    movel([0.255095, -1.387885, -2.566810, -0.757694, 1.570796, 1.825892],accel_mss,speed_ms,0,blend_radius_m)
    movel([0.255265, -1.387620, -2.567000, -0.757769, 1.570796, 1.826062],accel_mss,speed_ms,0,blend_radius_m)
    movel([0.255538, -1.387474, -2.567104, -0.757811, 1.570796, 1.826334],accel_mss,speed_ms,0,blend_radius_m)
    movel([0.255936, -1.387475, -2.567104, -0.757810, 1.570796, 1.826733],accel_mss,speed_ms,0,blend_radius_m)
    movel([0.256466, -1.387632, -2.566991, -0.757766, 1.570796, 1.827262],accel_mss,speed_ms,0,blend_radius_m)
    movel([0.257289, -1.388179, -2.566600, -0.757611, 1.570796, 1.828085],accel_mss,speed_ms,0,blend_radius_m)
    movel([0.257855, -1.389086, -2.565949, -0.757354, 1.570796, 1.828651],accel_mss,speed_ms,0,blend_radius_m)
    movel([0.258263, -1.390555, -2.564893, -0.756941, 1.570796, 1.829060],accel_mss,speed_ms,0,blend_radius_m)
    movel([0.259108, -1.396147, -2.560843, -0.755399, 1.570796, 1.829904],accel_mss,speed_ms,0,blend_radius_m)
    movel([0.259420, -1.397275, -2.560021, -0.755093, 1.570796, 1.830216],accel_mss,speed_ms,0,blend_radius_m)
    movel([0.259859, -1.398329, -2.559250, -0.754809, 1.570796, 1.830656],accel_mss,speed_ms,0,blend_radius_m)
    movel([0.260330, -1.399097, -2.558688, -0.754603, 1.570796, 1.831126],accel_mss,speed_ms,0,blend_radius_m)
    movel([0.260925, -1.399770, -2.558195, -0.754424, 1.570796, 1.831721],accel_mss,speed_ms,0,blend_radius_m)
    movel([0.261593, -1.400274, -2.557826, -0.754290, 1.570796, 1.832390],accel_mss,speed_ms,0,blend_radius_m)
    movel([0.262390, -1.400639, -2.557557, -0.754193, 1.570796, 1.833187],accel_mss,speed_ms,0,blend_radius_m)
    movel([0.263557, -1.400866, -2.557390, -0.754133, 1.570796, 1.834353],accel_mss,speed_ms,0,blend_radius_m)
    movel([0.264871, -1.400801, -2.557438, -0.754150, 1.570796, 1.835667],accel_mss,speed_ms,0,blend_radius_m)
    movel([0.266400, -1.400447, -2.557698, -0.754244, 1.570796, 1.837196],accel_mss,speed_ms,0,blend_radius_m)
    movel([0.267947, -1.399865, -2.558125, -0.754398, 1.570796, 1.838744],accel_mss,speed_ms,0,blend_radius_m)
    movel([0.269799, -1.398926, -2.558813, -0.754649, 1.570796, 1.840596],accel_mss,speed_ms,0,blend_radius_m)
    movel([0.271593, -1.397805, -2.559633, -0.754950, 1.570796, 1.842389],accel_mss,speed_ms,0,blend_radius_m)
    movel([0.273718, -1.396265, -2.560757, -0.755367, 1.570796, 1.844514],accel_mss,speed_ms,0,blend_radius_m)
    movel([0.276733, -1.393794, -2.562553, -0.756042, 1.570796, 1.847530],accel_mss,speed_ms,0,blend_radius_m)
    movel([0.277800, -1.392821, -2.563257, -0.756311, 1.570796, 1.848596],accel_mss,speed_ms,0,blend_radius_m)
    movel([0.279582, -1.391076, -2.564517, -0.756796, 1.570796, 1.850378],accel_mss,speed_ms,0,blend_radius_m)
    movel([0.281480, -1.388952, -2.566045, -0.757392, 1.570796, 1.852277],accel_mss,speed_ms,0,blend_radius_m)
    movel([0.283244, -1.386754, -2.567620, -0.758016, 1.570796, 1.854040],accel_mss,speed_ms,0,blend_radius_m)
    movel([0.285091, -1.384211, -2.569432, -0.758746, 1.570796, 1.855887],accel_mss,speed_ms,0,blend_radius_m)
    movel([0.286815, -1.381625, -2.571266, -0.759499, 1.570796, 1.857611],accel_mss,speed_ms,0,blend_radius_m)
    movel([0.288428, -1.378981, -2.573130, -0.760278, 1.570796, 1.859225],accel_mss,speed_ms,0,blend_radius_m)
    movel([0.289908, -1.376305, -2.575007, -0.761077, 1.570796, 1.860704],accel_mss,speed_ms,0,blend_radius_m)
    movel([0.291098, -1.373867, -2.576709, -0.761814, 1.570796, 1.861894],accel_mss,speed_ms,0,blend_radius_m)
    movel([0.292109, -1.371416, -2.578410, -0.762563, 1.570796, 1.862906],accel_mss,speed_ms,0,blend_radius_m)
    movel([0.292732, -1.369549, -2.579701, -0.763139, 1.570796, 1.863528],accel_mss,speed_ms,0,blend_radius_m)
    movel([0.293193, -1.367698, -2.580975, -0.763716, 1.570796, 1.863989],accel_mss,speed_ms,0,blend_radius_m)
    movel([0.293453, -1.365997, -2.582142, -0.764250, 1.570796, 1.864249],accel_mss,speed_ms,0,blend_radius_m)
    movel([0.293523, -1.364348, -2.583270, -0.764771, 1.570796, 1.864319],accel_mss,speed_ms,0,blend_radius_m)
    movel([0.293397, -1.362735, -2.584369, -0.765285, 1.570796, 1.864193],accel_mss,speed_ms,0,blend_radius_m)
    movel([0.293080, -1.361208, -2.585406, -0.765775, 1.570796, 1.863876],accel_mss,speed_ms,0,blend_radius_m)
    movel([0.292542, -1.359616, -2.586484, -0.766289, 1.570796, 1.863339],accel_mss,speed_ms,0,blend_radius_m)
    movel([0.291851, -1.358116, -2.587496, -0.766777, 1.570796, 1.862647],accel_mss,speed_ms,0,blend_radius_m)
    movel([0.290674, -1.356227, -2.588766, -0.767395, 1.570796, 1.861471],accel_mss,speed_ms,0,blend_radius_m)
    movel([0.290146, -1.355630, -2.589167, -0.767592, 1.570796, 1.860942],accel_mss,speed_ms,0,blend_radius_m)
    movel([0.289507, -1.355132, -2.589501, -0.767756, 1.570796, 1.860303],accel_mss,speed_ms,0,blend_radius_m)
    movel([0.288952, -1.354872, -2.589675, -0.767843, 1.570796, 1.859748],accel_mss,speed_ms,0,blend_radius_m)
    movel([0.288300, -1.354741, -2.589762, -0.767886, 1.570796, 1.859097],accel_mss,speed_ms,0,blend_radius_m)
    movel([0.287679, -1.354781, -2.589735, -0.767872, 1.570796, 1.858476],accel_mss,speed_ms,0,blend_radius_m)
    movel([0.287015, -1.355005, -2.589585, -0.767798, 1.570796, 1.857811],accel_mss,speed_ms,0,blend_radius_m)
    movel([0.286082, -1.355625, -2.589170, -0.767594, 1.570796, 1.856878],accel_mss,speed_ms,0,blend_radius_m)
    movel([0.285289, -1.356517, -2.588572, -0.767300, 1.570796, 1.856086],accel_mss,speed_ms,0,blend_radius_m)
    movel([0.284369, -1.358039, -2.587548, -0.766802, 1.570796, 1.855165],accel_mss,speed_ms,0,blend_radius_m)
    movel([0.282752, -1.361200, -2.585411, -0.765777, 1.570796, 1.853548],accel_mss,speed_ms,0,blend_radius_m)
    movel([0.280629, -1.365085, -2.582766, -0.764537, 1.570796, 1.851426],accel_mss,speed_ms,0,blend_radius_m)
    movel([0.278252, -1.368753, -2.580249, -0.763386, 1.570796, 1.849048],accel_mss,speed_ms,0,blend_radius_m)
    movel([0.275849, -1.371892, -2.578080, -0.762416, 1.570796, 1.846645],accel_mss,speed_ms,0,blend_radius_m)
    movel([0.274806, -1.373052, -2.577275, -0.762062, 1.570796, 1.845602],accel_mss,speed_ms,0,blend_radius_m)
    movel([0.272903, -1.374773, -2.576077, -0.761539, 1.570796, 1.843700],accel_mss,speed_ms,0,blend_radius_m)
    movel([0.272221, -1.375292, -2.575715, -0.761382, 1.570796, 1.843017],accel_mss,speed_ms,0,blend_radius_m)
    movel([0.270902, -1.376104, -2.575148, -0.761137, 1.570796, 1.841698],accel_mss,speed_ms,0,blend_radius_m)
    movel([0.270153, -1.376475, -2.574888, -0.761026, 1.570796, 1.840949],accel_mss,speed_ms,0,blend_radius_m)
    movel([0.269154, -1.376784, -2.574672, -0.760933, 1.570796, 1.839950],accel_mss,speed_ms,0,blend_radius_m)
    movel([0.268438, -1.376865, -2.574615, -0.760909, 1.570796, 1.839235],accel_mss,speed_ms,0,blend_radius_m)
    movel([0.267352, -1.376877, -2.574607, -0.760905, 1.570796, 1.838149],accel_mss,speed_ms,0,blend_radius_m)
    movel([0.267003, -1.376777, -2.574677, -0.760935, 1.570796, 1.837799],accel_mss,speed_ms,0,blend_radius_m)
    movel([0.266387, -1.376391, -2.574947, -0.761051, 1.570796, 1.837183],accel_mss,speed_ms,0,blend_radius_m)
    movel([0.266133, -1.376115, -2.575140, -0.761134, 1.570796, 1.836929],accel_mss,speed_ms,0,blend_radius_m)
    movel([0.265758, -1.375526, -2.575552, -0.761311, 1.570796, 1.836554],accel_mss,speed_ms,0,blend_radius_m)
    movel([0.265630, -1.375043, -2.575889, -0.761457, 1.570796, 1.836426],accel_mss,speed_ms,0,blend_radius_m)
    movel([0.265067, -1.369773, -2.579546, -0.763070, 1.570796, 1.835863],accel_mss,speed_ms,0,blend_radius_m)
    movel([0.264692, -1.365521, -2.582468, -0.764400, 1.570796, 1.835488],accel_mss,speed_ms,0,blend_radius_m)
    movel([0.263976, -1.360329, -2.586002, -0.766058, 1.570796, 1.834772],accel_mss,speed_ms,0,blend_radius_m)
    movel([0.263461, -1.358019, -2.587561, -0.766808, 1.570796, 1.834258],accel_mss,speed_ms,0,blend_radius_m)
    movel([0.262803, -1.355819, -2.589040, -0.767530, 1.570796, 1.833599],accel_mss,speed_ms,0,blend_radius_m)
    movel([0.261961, -1.353719, -2.590445, -0.768225, 1.570796, 1.832758],accel_mss,speed_ms,0,blend_radius_m)
    movel([0.261016, -1.351955, -2.591621, -0.768813, 1.570796, 1.831812],accel_mss,speed_ms,0,blend_radius_m)
    movel([0.259856, -1.350343, -2.592692, -0.769355, 1.570796, 1.830652],accel_mss,speed_ms,0,blend_radius_m)
    movel([0.258562, -1.348990, -2.593587, -0.769812, 1.570796, 1.829358],accel_mss,speed_ms,0,blend_radius_m)
    movel([0.257068, -1.347816, -2.594362, -0.770211, 1.570796, 1.827864],accel_mss,speed_ms,0,blend_radius_m)
    movel([0.255389, -1.346838, -2.595007, -0.770544, 1.570796, 1.826185],accel_mss,speed_ms,0,blend_radius_m)
    movel([0.253535, -1.346063, -2.595516, -0.770810, 1.570796, 1.824331],accel_mss,speed_ms,0,blend_radius_m)
    movel([0.252415, -1.345708, -2.595749, -0.770932, 1.570796, 1.823211],accel_mss,speed_ms,0,blend_radius_m)
    movel([0.251733, -1.345613, -2.595812, -0.770964, 1.570796, 1.822529],accel_mss,speed_ms,0,blend_radius_m)
    movel([0.251230, -1.345713, -2.595746, -0.770930, 1.570796, 1.822027],accel_mss,speed_ms,0,blend_radius_m)
    movel([0.250768, -1.346010, -2.595551, -0.770828, 1.570796, 1.821565],accel_mss,speed_ms,0,blend_radius_m)
    movel([0.250318, -1.346670, -2.595117, -0.770602, 1.570796, 1.821115],accel_mss,speed_ms,0,blend_radius_m)
    movel([0.249924, -1.348002, -2.594240, -0.770147, 1.570796, 1.820721],accel_mss,speed_ms,0,blend_radius_m)
    movel([0.249536, -1.349939, -2.592959, -0.769491, 1.570796, 1.820333],accel_mss,speed_ms,0,blend_radius_m)
    movel([0.249117, -1.352828, -2.591040, -0.768521, 1.570796, 1.819913],accel_mss,speed_ms,0,blend_radius_m)
    movel([0.248523, -1.356486, -2.588593, -0.767310, 1.570796, 1.819319],accel_mss,speed_ms,0,blend_radius_m)
    movel([0.248092, -1.358275, -2.587389, -0.766725, 1.570796, 1.818888],accel_mss,speed_ms,0,blend_radius_m)
    movel([0.246220, -1.365023, -2.582809, -0.764557, 1.570796, 1.817017],accel_mss,speed_ms,0,blend_radius_m)
    movel([0.245321, -1.367822, -2.580890, -0.763677, 1.570796, 1.816117],accel_mss,speed_ms,0,blend_radius_m)
    movel([0.242201, -1.375991, -2.575227, -0.761171, 1.570796, 1.812997],accel_mss,speed_ms,0,blend_radius_m)
    movel([0.239764, -1.381897, -2.571073, -0.759419, 1.570796, 1.810560],accel_mss,speed_ms,0,blend_radius_m)
    movel([0.237387, -1.387154, -2.567333, -0.757902, 1.570796, 1.808183],accel_mss,speed_ms,0,blend_radius_m)
    movel([0.235039, -1.391842, -2.563965, -0.756582, 1.570796, 1.805836],accel_mss,speed_ms,0,blend_radius_m)
    movel([0.231786, -1.397514, -2.559846, -0.755029, 1.570796, 1.802583],accel_mss,speed_ms,0,blend_radius_m)
    movel([0.231472, -1.397972, -2.559512, -0.754905, 1.570796, 1.802268],accel_mss,speed_ms,0,blend_radius_m)
    movel([0.231229, -1.398184, -2.559356, -0.754848, 1.570796, 1.802025],accel_mss,speed_ms,0,blend_radius_m)
    movel([0.230929, -1.398295, -2.559276, -0.754818, 1.570796, 1.801725],accel_mss,speed_ms,0,blend_radius_m)
    movel([0.230719, -1.398272, -2.559292, -0.754825, 1.570796, 1.801515],accel_mss,speed_ms,0,blend_radius_m)
    movel([0.230647, -1.398140, -2.559389, -0.754860, 1.570796, 1.801444],accel_mss,speed_ms,0,blend_radius_m)
    movel([0.231423, -1.395310, -2.561452, -0.755627, 1.570796, 1.802219],accel_mss,speed_ms,0,blend_radius_m)
    movel([0.231535, -1.394305, -2.562182, -0.755902, 1.570796, 1.802332],accel_mss,speed_ms,0,blend_radius_m)
    movel([0.231433, -1.393186, -2.562993, -0.756210, 1.570796, 1.802229],accel_mss,speed_ms,0,blend_radius_m)
    movel([0.231036, -1.391255, -2.564388, -0.756746, 1.570796, 1.801833],accel_mss,speed_ms,0,blend_radius_m)
    movel([0.230646, -1.388956, -2.566042, -0.757391, 1.570796, 1.801443],accel_mss,speed_ms,0,blend_radius_m)
    movel([0.230572, -1.386887, -2.567524, -0.757978, 1.570796, 1.801369],accel_mss,speed_ms,0,blend_radius_m)
    movel([0.230812, -1.384183, -2.569452, -0.758754, 1.570796, 1.801608],accel_mss,speed_ms,0,blend_radius_m)
    movel([0.231528, -1.379286, -2.572916, -0.760188, 1.570796, 1.802324],accel_mss,speed_ms,0,blend_radius_m)
    movel([0.232292, -1.373125, -2.577225, -0.762040, 1.570796, 1.803089],accel_mss,speed_ms,0,blend_radius_m)
    movel([0.232470, -1.370485, -2.579054, -0.762850, 1.570796, 1.803266],accel_mss,speed_ms,0,blend_radius_m)
    movel([0.232513, -1.367882, -2.580849, -0.763658, 1.570796, 1.803309],accel_mss,speed_ms,0,blend_radius_m)
    movel([0.232417, -1.365596, -2.582417, -0.764376, 1.570796, 1.803213],accel_mss,speed_ms,0,blend_radius_m)
    movel([0.232184, -1.363359, -2.583944, -0.765086, 1.570796, 1.802980],accel_mss,speed_ms,0,blend_radius_m)
    movel([0.231819, -1.361328, -2.585325, -0.765736, 1.570796, 1.802616],accel_mss,speed_ms,0,blend_radius_m)
    movel([0.231292, -1.359376, -2.586646, -0.766367, 1.570796, 1.802088],accel_mss,speed_ms,0,blend_radius_m)
    movel([0.230545, -1.357337, -2.588021, -0.767031, 1.570796, 1.801342],accel_mss,speed_ms,0,blend_radius_m)
    movel([0.229699, -1.355644, -2.589158, -0.767588, 1.570796, 1.800495],accel_mss,speed_ms,0,blend_radius_m)
    movel([0.228650, -1.354120, -2.590177, -0.768091, 1.570796, 1.799447],accel_mss,speed_ms,0,blend_radius_m)
    movel([0.227292, -1.352590, -2.591198, -0.768601, 1.570796, 1.798088],accel_mss,speed_ms,0,blend_radius_m)
    movel([0.225840, -1.351336, -2.592032, -0.769021, 1.570796, 1.796636],accel_mss,speed_ms,0,blend_radius_m)
    movel([0.224294, -1.350424, -2.592638, -0.769327, 1.570796, 1.795090],accel_mss,speed_ms,0,blend_radius_m)
    movel([0.222638, -1.349849, -2.593019, -0.769521, 1.570796, 1.793435],accel_mss,speed_ms,0,blend_radius_m)
    movel([0.220857, -1.349600, -2.593184, -0.769605, 1.570796, 1.791653],accel_mss,speed_ms,0,blend_radius_m)
    movel([0.219370, -1.349643, -2.593155, -0.769591, 1.570796, 1.790166],accel_mss,speed_ms,0,blend_radius_m)
    movel([0.217805, -1.349909, -2.592979, -0.769501, 1.570796, 1.788601],accel_mss,speed_ms,0,blend_radius_m)
    movel([0.216251, -1.350382, -2.592666, -0.769342, 1.570796, 1.787048],accel_mss,speed_ms,0,blend_radius_m)
    movel([0.214697, -1.351068, -2.592211, -0.769111, 1.570796, 1.785493],accel_mss,speed_ms,0,blend_radius_m)
    movel([0.213185, -1.351948, -2.591625, -0.768815, 1.570796, 1.783981],accel_mss,speed_ms,0,blend_radius_m)
    movel([0.211756, -1.352999, -2.590926, -0.768464, 1.570796, 1.782553],accel_mss,speed_ms,0,blend_radius_m)
    movel([0.210399, -1.354224, -2.590108, -0.768057, 1.570796, 1.781195],accel_mss,speed_ms,0,blend_radius_m)
    movel([0.208813, -1.356025, -2.588902, -0.767462, 1.570796, 1.779609],accel_mss,speed_ms,0,blend_radius_m)
    movel([0.208461, -1.356503, -2.588581, -0.767305, 1.570796, 1.779257],accel_mss,speed_ms,0,blend_radius_m)
    movel([0.207795, -1.357594, -2.587848, -0.766947, 1.570796, 1.778591],accel_mss,speed_ms,0,blend_radius_m)
    movel([0.207515, -1.357910, -2.587635, -0.766844, 1.570796, 1.778311],accel_mss,speed_ms,0,blend_radius_m)
    movel([0.207218, -1.358097, -2.587509, -0.766783, 1.570796, 1.778014],accel_mss,speed_ms,0,blend_radius_m)
    movel([0.206945, -1.358140, -2.587480, -0.766769, 1.570796, 1.777741],accel_mss,speed_ms,0,blend_radius_m)
    movel([0.206737, -1.357986, -2.587584, -0.766819, 1.570796, 1.777533],accel_mss,speed_ms,0,blend_radius_m)
    movel([0.206764, -1.357690, -2.587783, -0.766916, 1.570796, 1.777560],accel_mss,speed_ms,0,blend_radius_m)
    movel([0.207503, -1.356392, -2.588655, -0.767341, 1.570796, 1.778299],accel_mss,speed_ms,0,blend_radius_m)
    movel([0.208775, -1.354760, -2.589750, -0.767879, 1.570796, 1.779572],accel_mss,speed_ms,0,blend_radius_m)
    movel([0.210327, -1.353184, -2.590803, -0.768403, 1.570796, 1.781123],accel_mss,speed_ms,0,blend_radius_m)
    movel([0.211548, -1.352151, -2.591491, -0.768748, 1.570796, 1.782344],accel_mss,speed_ms,0,blend_radius_m)
    movel([0.212843, -1.351218, -2.592111, -0.769060, 1.570796, 1.783639],accel_mss,speed_ms,0,blend_radius_m)
    movel([0.214163, -1.350420, -2.592640, -0.769329, 1.570796, 1.784959],accel_mss,speed_ms,0,blend_radius_m)
    movel([0.215522, -1.349753, -2.593082, -0.769554, 1.570796, 1.786318],accel_mss,speed_ms,0,blend_radius_m)
    movel([0.216900, -1.349227, -2.593431, -0.769732, 1.570796, 1.787696],accel_mss,speed_ms,0,blend_radius_m)
    movel([0.218268, -1.348854, -2.593677, -0.769858, 1.570796, 1.789065],accel_mss,speed_ms,0,blend_radius_m)
    movel([0.219652, -1.348624, -2.593829, -0.769936, 1.570796, 1.790448],accel_mss,speed_ms,0,blend_radius_m)
    movel([0.220986, -1.348545, -2.593881, -0.769963, 1.570796, 1.791782],accel_mss,speed_ms,0,blend_radius_m)
    movel([0.222782, -1.348704, -2.593776, -0.769909, 1.570796, 1.793578],accel_mss,speed_ms,0,blend_radius_m)
    movel([0.224379, -1.349179, -2.593462, -0.769748, 1.570796, 1.795175],accel_mss,speed_ms,0,blend_radius_m)
    movel([0.226051, -1.350036, -2.592895, -0.769458, 1.570796, 1.796847],accel_mss,speed_ms,0,blend_radius_m)
    movel([0.227532, -1.351097, -2.592191, -0.769101, 1.570796, 1.798328],accel_mss,speed_ms,0,blend_radius_m)
    movel([0.228968, -1.352491, -2.591264, -0.768634, 1.570796, 1.799764],accel_mss,speed_ms,0,blend_radius_m)
    movel([0.230183, -1.354068, -2.590212, -0.768109, 1.570796, 1.800979],accel_mss,speed_ms,0,blend_radius_m)
    movel([0.231241, -1.355893, -2.588990, -0.767505, 1.570796, 1.802037],accel_mss,speed_ms,0,blend_radius_m)
    movel([0.232082, -1.357856, -2.587671, -0.766862, 1.570796, 1.802878],accel_mss,speed_ms,0,blend_radius_m)
    movel([0.232741, -1.360024, -2.586208, -0.766157, 1.570796, 1.803537],accel_mss,speed_ms,0,blend_radius_m)
    movel([0.233194, -1.362294, -2.584669, -0.765426, 1.570796, 1.803990],accel_mss,speed_ms,0,blend_radius_m)
    movel([0.233471, -1.364806, -2.582957, -0.764626, 1.570796, 1.804267],accel_mss,speed_ms,0,blend_radius_m)
    movel([0.233565, -1.367384, -2.581191, -0.763814, 1.570796, 1.804361],accel_mss,speed_ms,0,blend_radius_m)
    movel([0.233479, -1.370501, -2.579043, -0.762845, 1.570796, 1.804275],accel_mss,speed_ms,0,blend_radius_m)
    movel([0.233220, -1.373662, -2.576851, -0.761876, 1.570796, 1.804017],accel_mss,speed_ms,0,blend_radius_m)
    movel([0.232141, -1.381784, -2.571153, -0.759452, 1.570796, 1.802937],accel_mss,speed_ms,0,blend_radius_m)
    movel([0.231723, -1.384753, -2.569046, -0.758590, 1.570796, 1.802520],accel_mss,speed_ms,0,blend_radius_m)
    movel([0.231587, -1.386705, -2.567654, -0.758030, 1.570796, 1.802384],accel_mss,speed_ms,0,blend_radius_m)
    movel([0.231680, -1.388416, -2.566430, -0.757543, 1.570796, 1.802476],accel_mss,speed_ms,0,blend_radius_m)
    movel([0.232016, -1.390502, -2.564931, -0.756956, 1.570796, 1.802813],accel_mss,speed_ms,0,blend_radius_m)
    movel([0.232538, -1.393687, -2.562630, -0.756072, 1.570796, 1.803334],accel_mss,speed_ms,0,blend_radius_m)
    movel([0.232642, -1.394026, -2.562384, -0.755978, 1.570796, 1.803438],accel_mss,speed_ms,0,blend_radius_m)
    movel([0.232836, -1.393978, -2.562419, -0.755992, 1.570796, 1.803633],accel_mss,speed_ms,0,blend_radius_m)
    movel([0.233230, -1.393353, -2.562872, -0.756164, 1.570796, 1.804026],accel_mss,speed_ms,0,blend_radius_m)
    movel([0.237057, -1.385694, -2.568376, -0.758319, 1.570796, 1.807853],accel_mss,speed_ms,0,blend_radius_m)
    movel([0.239796, -1.379520, -2.572750, -0.760118, 1.570796, 1.810592],accel_mss,speed_ms,0,blend_radius_m)
    movel([0.242407, -1.373049, -2.577278, -0.762063, 1.570796, 1.813204],accel_mss,speed_ms,0,blend_radius_m)
    movel([0.244761, -1.366579, -2.581744, -0.764067, 1.570796, 1.815557],accel_mss,speed_ms,0,blend_radius_m)
    movel([0.245773, -1.363351, -2.583950, -0.765088, 1.570796, 1.816569],accel_mss,speed_ms,0,blend_radius_m)
    movel([0.246728, -1.359698, -2.586428, -0.766263, 1.570796, 1.817525],accel_mss,speed_ms,0,blend_radius_m)
    movel([0.247527, -1.356058, -2.588880, -0.767451, 1.570796, 1.818323],accel_mss,speed_ms,0,blend_radius_m)
    movel([0.248051, -1.352879, -2.591005, -0.768504, 1.570796, 1.818848],accel_mss,speed_ms,0,blend_radius_m)
    movel([0.248446, -1.350238, -2.592761, -0.769390, 1.570796, 1.819242],accel_mss,speed_ms,0,blend_radius_m)
    movel([0.248857, -1.348235, -2.594086, -0.770068, 1.570796, 1.819653],accel_mss,speed_ms,0,blend_radius_m)
    movel([0.249288, -1.346744, -2.595068, -0.770577, 1.570796, 1.820084],accel_mss,speed_ms,0,blend_radius_m)
    movel([0.249754, -1.345882, -2.595635, -0.770872, 1.570796, 1.820550],accel_mss,speed_ms,0,blend_radius_m)
    movel([0.250249, -1.345323, -2.596002, -0.771064, 1.570796, 1.821045],accel_mss,speed_ms,0,blend_radius_m)
    movel([0.250776, -1.344913, -2.596271, -0.771205, 1.570796, 1.821572],accel_mss,speed_ms,0,blend_radius_m)
    movel([0.251321, -1.344661, -2.596436, -0.771292, 1.570796, 1.822117],accel_mss,speed_ms,0,blend_radius_m)
    movel([0.251873, -1.344569, -2.596497, -0.771324, 1.570796, 1.822669],accel_mss,speed_ms,0,blend_radius_m)
    movel([0.252588, -1.344649, -2.596444, -0.771296, 1.570796, 1.823385],accel_mss,speed_ms,0,blend_radius_m)
    movel([0.253955, -1.345029, -2.596195, -0.771165, 1.570796, 1.824751],accel_mss,speed_ms,0,blend_radius_m)
    movel([0.256341, -1.345925, -2.595607, -0.770857, 1.570796, 1.827138],accel_mss,speed_ms,0,blend_radius_m)
    movel([0.258315, -1.347164, -2.594792, -0.770433, 1.570796, 1.829111],accel_mss,speed_ms,0,blend_radius_m)
    movel([0.260118, -1.348786, -2.593722, -0.769881, 1.570796, 1.830914],accel_mss,speed_ms,0,blend_radius_m)
    movel([0.261674, -1.350714, -2.592445, -0.769230, 1.570796, 1.832470],accel_mss,speed_ms,0,blend_radius_m)
    movel([0.262915, -1.352863, -2.591016, -0.768509, 1.570796, 1.833711],accel_mss,speed_ms,0,blend_radius_m)
    movel([0.263612, -1.354489, -2.589931, -0.767969, 1.570796, 1.834408],accel_mss,speed_ms,0,blend_radius_m)
    movel([0.264185, -1.356184, -2.588795, -0.767410, 1.570796, 1.834981],accel_mss,speed_ms,0,blend_radius_m)
    movel([0.265108, -1.360143, -2.586127, -0.766118, 1.570796, 1.835905],accel_mss,speed_ms,0,blend_radius_m)
    movel([0.265810, -1.365284, -2.582630, -0.764475, 1.570796, 1.836606],accel_mss,speed_ms,0,blend_radius_m)
    movel([0.266385, -1.372378, -2.577743, -0.762268, 1.570796, 1.837182],accel_mss,speed_ms,0,blend_radius_m)
    movel([0.266613, -1.374304, -2.576404, -0.761681, 1.570796, 1.837409],accel_mss,speed_ms,0,blend_radius_m)
    movel([0.266771, -1.374866, -2.576012, -0.761511, 1.570796, 1.837568],accel_mss,speed_ms,0,blend_radius_m)
    movel([0.267041, -1.375360, -2.575667, -0.761361, 1.570796, 1.837837],accel_mss,speed_ms,0,blend_radius_m)
    movel([0.267347, -1.375658, -2.575460, -0.761272, 1.570796, 1.838143],accel_mss,speed_ms,0,blend_radius_m)
    movel([0.267760, -1.375844, -2.575329, -0.761215, 1.570796, 1.838556],accel_mss,speed_ms,0,blend_radius_m)
    movel([0.268285, -1.375927, -2.575272, -0.761191, 1.570796, 1.839082],accel_mss,speed_ms,0,blend_radius_m)
    movel([0.268867, -1.375899, -2.575291, -0.761199, 1.570796, 1.839663],accel_mss,speed_ms,0,blend_radius_m)
    movel([0.269616, -1.375740, -2.575402, -0.761247, 1.570796, 1.840412],accel_mss,speed_ms,0,blend_radius_m)
    movel([0.270377, -1.375462, -2.575596, -0.761331, 1.570796, 1.841174],accel_mss,speed_ms,0,blend_radius_m)
    movel([0.271129, -1.375077, -2.575865, -0.761447, 1.570796, 1.841925],accel_mss,speed_ms,0,blend_radius_m)
    movel([0.271844, -1.374596, -2.576200, -0.761592, 1.570796, 1.842640],accel_mss,speed_ms,0,blend_radius_m)
    movel([0.273576, -1.373133, -2.577219, -0.762037, 1.570796, 1.844373],accel_mss,speed_ms,0,blend_radius_m)
    movel([0.275126, -1.371513, -2.578343, -0.762533, 1.570796, 1.845922],accel_mss,speed_ms,0,blend_radius_m)
    movel([0.276981, -1.369177, -2.579957, -0.763255, 1.570796, 1.847777],accel_mss,speed_ms,0,blend_radius_m)
    movel([0.278604, -1.366757, -2.581622, -0.764011, 1.570796, 1.849400],accel_mss,speed_ms,0,blend_radius_m)
    movel([0.280459, -1.363589, -2.583787, -0.765012, 1.570796, 1.851256],accel_mss,speed_ms,0,blend_radius_m)
    movel([0.283390, -1.357989, -2.587582, -0.766818, 1.570796, 1.854186],accel_mss,speed_ms,0,blend_radius_m)
    movel([0.284147, -1.356672, -2.588468, -0.767249, 1.570796, 1.854944],accel_mss,speed_ms,0,blend_radius_m)
    movel([0.284772, -1.355802, -2.589051, -0.767535, 1.570796, 1.855569],accel_mss,speed_ms,0,blend_radius_m)
    movel([0.285460, -1.355101, -2.589521, -0.767767, 1.570796, 1.856256],accel_mss,speed_ms,0,blend_radius_m)
    movel([0.286130, -1.354583, -2.589868, -0.767938, 1.570796, 1.856926],accel_mss,speed_ms,0,blend_radius_m)
    movel([0.286753, -1.354223, -2.590108, -0.768057, 1.570796, 1.857549],accel_mss,speed_ms,0,blend_radius_m)
    movel([0.287401, -1.353985, -2.590268, -0.768136, 1.570796, 1.858197],accel_mss,speed_ms,0,blend_radius_m)
    movel([0.288149, -1.353838, -2.590366, -0.768185, 1.570796, 1.858946],accel_mss,speed_ms,0,blend_radius_m)
    movel([0.288852, -1.353812, -2.590383, -0.768194, 1.570796, 1.859649],accel_mss,speed_ms,0,blend_radius_m)
    movel([0.289487, -1.353922, -2.590310, -0.768157, 1.570796, 1.860283],accel_mss,speed_ms,0,blend_radius_m)
    movel([0.290701, -1.354530, -2.589903, -0.767956, 1.570796, 1.861497],accel_mss,speed_ms,0,blend_radius_m)
    movel([0.291837, -1.355686, -2.589129, -0.767574, 1.570796, 1.862634],accel_mss,speed_ms,0,blend_radius_m)
    movel([0.292934, -1.357455, -2.587941, -0.766993, 1.570796, 1.863730],accel_mss,speed_ms,0,blend_radius_m)
    movel([0.293974, -1.359880, -2.586306, -0.766204, 1.570796, 1.864770],accel_mss,speed_ms,0,blend_radius_m)
    movel([0.294523, -1.362239, -2.584706, -0.765444, 1.570796, 1.865319],accel_mss,speed_ms,0,blend_radius_m)
    movel([0.294624, -1.363458, -2.583877, -0.765054, 1.570796, 1.865420],accel_mss,speed_ms,0,blend_radius_m)
    movel([0.294609, -1.364722, -2.583014, -0.764653, 1.570796, 1.865406],accel_mss,speed_ms,0,blend_radius_m)
    movel([0.294266, -1.367507, -2.581107, -0.763775, 1.570796, 1.865062],accel_mss,speed_ms,0,blend_radius_m)
    movel([0.293918, -1.368891, -2.580154, -0.763344, 1.570796, 1.864714],accel_mss,speed_ms,0,blend_radius_m)
    movel([0.293268, -1.370843, -2.578807, -0.762739, 1.570796, 1.864064],accel_mss,speed_ms,0,blend_radius_m)
    movel([0.291751, -1.374603, -2.576196, -0.761590, 1.570796, 1.862547],accel_mss,speed_ms,0,blend_radius_m)
    movel([0.290553, -1.376888, -2.574599, -0.760902, 1.570796, 1.861349],accel_mss,speed_ms,0,blend_radius_m)
    speed_ms = 0.005
    movel([0.290553, -1.368165, -2.570582, -0.773641, 1.570796, 1.861349],accel_mss,speed_ms,0,blend_radius_m)
    speed_ms = 0.040
    movel([0.320654, -1.348290, -2.584044, -0.780055, 1.570796, 1.891451],accel_mss,speed_ms,0,blend_radius_m)
    speed_ms = 0.005
    movel([0.320654, -1.357148, -2.588148, -0.767093, 1.570796, 1.891451],accel_mss,speed_ms,0,blend_radius_m)
    speed_ms = 0.025
    movel([0.319732, -1.357074, -2.588198, -0.767118, 1.570796, 1.890528],accel_mss,speed_ms,0,blend_radius_m)
    movel([0.319205, -1.356915, -2.588304, -0.767170, 1.570796, 1.890001],accel_mss,speed_ms,0,blend_radius_m)
    movel([0.317857, -1.356295, -2.588721, -0.767373, 1.570796, 1.888654],accel_mss,speed_ms,0,blend_radius_m)
    movel([0.317320, -1.355922, -2.588971, -0.767496, 1.570796, 1.888117],accel_mss,speed_ms,0,blend_radius_m)
    movel([0.316201, -1.354707, -2.589785, -0.767897, 1.570796, 1.886997],accel_mss,speed_ms,0,blend_radius_m)
    movel([0.314823, -1.352667, -2.591147, -0.768575, 1.570796, 1.885619],accel_mss,speed_ms,0,blend_radius_m)
    movel([0.313237, -1.349704, -2.593115, -0.769570, 1.570796, 1.884034],accel_mss,speed_ms,0,blend_radius_m)
    movel([0.311845, -1.346731, -2.595077, -0.770581, 1.570796, 1.882641],accel_mss,speed_ms,0,blend_radius_m)
    movel([0.311446, -1.345137, -2.596124, -0.771128, 1.570796, 1.882243],accel_mss,speed_ms,0,blend_radius_m)
    movel([0.311462, -1.344439, -2.596581, -0.771368, 1.570796, 1.882258],accel_mss,speed_ms,0,blend_radius_m)
    movel([0.312033, -1.342330, -2.597959, -0.772099, 1.570796, 1.882830],accel_mss,speed_ms,0,blend_radius_m)
    movel([0.313181, -1.338985, -2.600133, -0.773272, 1.570796, 1.883977],accel_mss,speed_ms,0,blend_radius_m)
    movel([0.315208, -1.333366, -2.603748, -0.775275, 1.570796, 1.886004],accel_mss,speed_ms,0,blend_radius_m)
    movel([0.316058, -1.331299, -2.605067, -0.776022, 1.570796, 1.886855],accel_mss,speed_ms,0,blend_radius_m)
    movel([0.317881, -1.327107, -2.607725, -0.777556, 1.570796, 1.888677],accel_mss,speed_ms,0,blend_radius_m)
    movel([0.318194, -1.326115, -2.608351, -0.777923, 1.570796, 1.888990],accel_mss,speed_ms,0,blend_radius_m)
    movel([0.318267, -1.325423, -2.608786, -0.778179, 1.570796, 1.889064],accel_mss,speed_ms,0,blend_radius_m)
    movel([0.318110, -1.324962, -2.609077, -0.778351, 1.570796, 1.888907],accel_mss,speed_ms,0,blend_radius_m)
    movel([0.317737, -1.324753, -2.609207, -0.778428, 1.570796, 1.888533],accel_mss,speed_ms,0,blend_radius_m)
    movel([0.317436, -1.324772, -2.609196, -0.778421, 1.570796, 1.888233],accel_mss,speed_ms,0,blend_radius_m)
    movel([0.316115, -1.325001, -2.609052, -0.778336, 1.570796, 1.886911],accel_mss,speed_ms,0,blend_radius_m)
    movel([0.315993, -1.324904, -2.609113, -0.778372, 1.570796, 1.886790],accel_mss,speed_ms,0,blend_radius_m)
    movel([0.315921, -1.324400, -2.609429, -0.778560, 1.570796, 1.886717],accel_mss,speed_ms,0,blend_radius_m)
    movel([0.315980, -1.324129, -2.609599, -0.778661, 1.570796, 1.886777],accel_mss,speed_ms,0,blend_radius_m)
    movel([0.317198, -1.321892, -2.610999, -0.779498, 1.570796, 1.887995],accel_mss,speed_ms,0,blend_radius_m)
    movel([0.317469, -1.321421, -2.611293, -0.779675, 1.570796, 1.888265],accel_mss,speed_ms,0,blend_radius_m)
    movel([0.318083, -1.320351, -2.611960, -0.780079, 1.570796, 1.888879],accel_mss,speed_ms,0,blend_radius_m)
    movel([0.315622, -1.322333, -2.610723, -0.779332, 1.570796, 1.886419],accel_mss,speed_ms,0,blend_radius_m)
    movel([0.313339, -1.324104, -2.609615, -0.778670, 1.570796, 1.884135],accel_mss,speed_ms,0,blend_radius_m)
    movel([0.310995, -1.325778, -2.608563, -0.778048, 1.570796, 1.881791],accel_mss,speed_ms,0,blend_radius_m)
    movel([0.308638, -1.327328, -2.607586, -0.777475, 1.570796, 1.879434],accel_mss,speed_ms,0,blend_radius_m)
    movel([0.306302, -1.328723, -2.606703, -0.776962, 1.570796, 1.877099],accel_mss,speed_ms,0,blend_radius_m)
    movel([0.304835, -1.329490, -2.606218, -0.776682, 1.570796, 1.875632],accel_mss,speed_ms,0,blend_radius_m)
    movel([0.304548, -1.329552, -2.606178, -0.776659, 1.570796, 1.875345],accel_mss,speed_ms,0,blend_radius_m)
    movel([0.304344, -1.329458, -2.606238, -0.776693, 1.570796, 1.875141],accel_mss,speed_ms,0,blend_radius_m)
    movel([0.304305, -1.329242, -2.606375, -0.776772, 1.570796, 1.875101],accel_mss,speed_ms,0,blend_radius_m)
    movel([0.304442, -1.328987, -2.606536, -0.776866, 1.570796, 1.875238],accel_mss,speed_ms,0,blend_radius_m)
    movel([0.305573, -1.327819, -2.607276, -0.777294, 1.570796, 1.876370],accel_mss,speed_ms,0,blend_radius_m)
    movel([0.307878, -1.325397, -2.608803, -0.778189, 1.570796, 1.878674],accel_mss,speed_ms,0,blend_radius_m)
    movel([0.308860, -1.324183, -2.609565, -0.778641, 1.570796, 1.879657],accel_mss,speed_ms,0,blend_radius_m)
    movel([0.310446, -1.321890, -2.611000, -0.779499, 1.570796, 1.881243],accel_mss,speed_ms,0,blend_radius_m)
    movel([0.310222, -1.321875, -2.611010, -0.779504, 1.570796, 1.881019],accel_mss,speed_ms,0,blend_radius_m)
    movel([0.308575, -1.323006, -2.610303, -0.779080, 1.570796, 1.879372],accel_mss,speed_ms,0,blend_radius_m)
    movel([0.301104, -1.327684, -2.607361, -0.777344, 1.570796, 1.871900],accel_mss,speed_ms,0,blend_radius_m)
    movel([0.299050, -1.329068, -2.606485, -0.776836, 1.570796, 1.869847],accel_mss,speed_ms,0,blend_radius_m)
    movel([0.297441, -1.330295, -2.605706, -0.776388, 1.570796, 1.868237],accel_mss,speed_ms,0,blend_radius_m)
    movel([0.296047, -1.331530, -2.604920, -0.775939, 1.570796, 1.866843],accel_mss,speed_ms,0,blend_radius_m)
    movel([0.294685, -1.332763, -2.604133, -0.775492, 1.570796, 1.865481],accel_mss,speed_ms,0,blend_radius_m)
    movel([0.294292, -1.332618, -2.604226, -0.775545, 1.570796, 1.865088],accel_mss,speed_ms,0,blend_radius_m)
    movel([0.294286, -1.332414, -2.604357, -0.775619, 1.570796, 1.865082],accel_mss,speed_ms,0,blend_radius_m)
    movel([0.294844, -1.331341, -2.605041, -0.776007, 1.570796, 1.865640],accel_mss,speed_ms,0,blend_radius_m)
    movel([0.295532, -1.330237, -2.605743, -0.776409, 1.570796, 1.866328],accel_mss,speed_ms,0,blend_radius_m)
    movel([0.297118, -1.327651, -2.607382, -0.777356, 1.570796, 1.867914],accel_mss,speed_ms,0,blend_radius_m)
    movel([0.297456, -1.327008, -2.607788, -0.777593, 1.570796, 1.868252],accel_mss,speed_ms,0,blend_radius_m)
    movel([0.297392, -1.326908, -2.607851, -0.777630, 1.570796, 1.868188],accel_mss,speed_ms,0,blend_radius_m)
    movel([0.294597, -1.329026, -2.606512, -0.776851, 1.570796, 1.865393],accel_mss,speed_ms,0,blend_radius_m)
    movel([0.294232, -1.329233, -2.606381, -0.776776, 1.570796, 1.865029],accel_mss,speed_ms,0,blend_radius_m)
    movel([0.293693, -1.329365, -2.606297, -0.776727, 1.570796, 1.864490],accel_mss,speed_ms,0,blend_radius_m)
    movel([0.293346, -1.329649, -2.606116, -0.776623, 1.570796, 1.864143],accel_mss,speed_ms,0,blend_radius_m)
    movel([0.291598, -1.331921, -2.604671, -0.775797, 1.570796, 1.862395],accel_mss,speed_ms,0,blend_radius_m)
    movel([0.290405, -1.333593, -2.603603, -0.775193, 1.570796, 1.861201],accel_mss,speed_ms,0,blend_radius_m)
    movel([0.287976, -1.337290, -2.601228, -0.773871, 1.570796, 1.858773],accel_mss,speed_ms,0,blend_radius_m)
    movel([0.287961, -1.337510, -2.601086, -0.773793, 1.570796, 1.858758],accel_mss,speed_ms,0,blend_radius_m)
    movel([0.288199, -1.337535, -2.601070, -0.773785, 1.570796, 1.858995],accel_mss,speed_ms,0,blend_radius_m)
    movel([0.290317, -1.336686, -2.601617, -0.774086, 1.570796, 1.861113],accel_mss,speed_ms,0,blend_radius_m)
    movel([0.293851, -1.335132, -2.602617, -0.774641, 1.570796, 1.864647],accel_mss,speed_ms,0,blend_radius_m)
    movel([0.294956, -1.334603, -2.602956, -0.774830, 1.570796, 1.865753],accel_mss,speed_ms,0,blend_radius_m)
    movel([0.295611, -1.334390, -2.603093, -0.774907, 1.570796, 1.866407],accel_mss,speed_ms,0,blend_radius_m)
    movel([0.295912, -1.334448, -2.603055, -0.774886, 1.570796, 1.866708],accel_mss,speed_ms,0,blend_radius_m)
    movel([0.295964, -1.334711, -2.602887, -0.774791, 1.570796, 1.866761],accel_mss,speed_ms,0,blend_radius_m)
    movel([0.295755, -1.335062, -2.602661, -0.774666, 1.570796, 1.866551],accel_mss,speed_ms,0,blend_radius_m)
    movel([0.295404, -1.335329, -2.602490, -0.774570, 1.570796, 1.866201],accel_mss,speed_ms,0,blend_radius_m)
    movel([0.292890, -1.336544, -2.601708, -0.774136, 1.570796, 1.863687],accel_mss,speed_ms,0,blend_radius_m)
    movel([0.290019, -1.337759, -2.600925, -0.773705, 1.570796, 1.860816],accel_mss,speed_ms,0,blend_radius_m)
    movel([0.287226, -1.338734, -2.600295, -0.773360, 1.570796, 1.858022],accel_mss,speed_ms,0,blend_radius_m)
    movel([0.285045, -1.339277, -2.599943, -0.773169, 1.570796, 1.855842],accel_mss,speed_ms,0,blend_radius_m)
    movel([0.282043, -1.339775, -2.599621, -0.772994, 1.570796, 1.852840],accel_mss,speed_ms,0,blend_radius_m)
    movel([0.279156, -1.340130, -2.599391, -0.772869, 1.570796, 1.849953],accel_mss,speed_ms,0,blend_radius_m)
    movel([0.277660, -1.340102, -2.599409, -0.772879, 1.570796, 1.848456],accel_mss,speed_ms,0,blend_radius_m)
    movel([0.277015, -1.339943, -2.599511, -0.772934, 1.570796, 1.847812],accel_mss,speed_ms,0,blend_radius_m)
    movel([0.276671, -1.339700, -2.599669, -0.773020, 1.570796, 1.847467],accel_mss,speed_ms,0,blend_radius_m)
    movel([0.276612, -1.339378, -2.599878, -0.773133, 1.570796, 1.847408],accel_mss,speed_ms,0,blend_radius_m)
    movel([0.276808, -1.338983, -2.600133, -0.773272, 1.570796, 1.847605],accel_mss,speed_ms,0,blend_radius_m)
    movel([0.277370, -1.338634, -2.600360, -0.773396, 1.570796, 1.848167],accel_mss,speed_ms,0,blend_radius_m)
    movel([0.277906, -1.338486, -2.600455, -0.773448, 1.570796, 1.848702],accel_mss,speed_ms,0,blend_radius_m)
    movel([0.280351, -1.337938, -2.600809, -0.773642, 1.570796, 1.851147],accel_mss,speed_ms,0,blend_radius_m)
    movel([0.281641, -1.337503, -2.601090, -0.773796, 1.570796, 1.852437],accel_mss,speed_ms,0,blend_radius_m)
    movel([0.282913, -1.336923, -2.601464, -0.774002, 1.570796, 1.853710],accel_mss,speed_ms,0,blend_radius_m)
    movel([0.284303, -1.336137, -2.601970, -0.774282, 1.570796, 1.855100],accel_mss,speed_ms,0,blend_radius_m)
    movel([0.285149, -1.335647, -2.602286, -0.774457, 1.570796, 1.855945],accel_mss,speed_ms,0,blend_radius_m)
    movel([0.285592, -1.335482, -2.602392, -0.774515, 1.570796, 1.856388],accel_mss,speed_ms,0,blend_radius_m)
    movel([0.285779, -1.335562, -2.602340, -0.774487, 1.570796, 1.856575],accel_mss,speed_ms,0,blend_radius_m)
    movel([0.285771, -1.335855, -2.602152, -0.774382, 1.570796, 1.856568],accel_mss,speed_ms,0,blend_radius_m)
    movel([0.285413, -1.336346, -2.601836, -0.774207, 1.570796, 1.856209],accel_mss,speed_ms,0,blend_radius_m)
    movel([0.284464, -1.337016, -2.601404, -0.773969, 1.570796, 1.855260],accel_mss,speed_ms,0,blend_radius_m)
    movel([0.283131, -1.337769, -2.600918, -0.773701, 1.570796, 1.853927],accel_mss,speed_ms,0,blend_radius_m)
    movel([0.281471, -1.338553, -2.600412, -0.773424, 1.570796, 1.852268],accel_mss,speed_ms,0,blend_radius_m)
    movel([0.280164, -1.339128, -2.600040, -0.773221, 1.570796, 1.850960],accel_mss,speed_ms,0,blend_radius_m)
    movel([0.283183, -1.338620, -2.600369, -0.773400, 1.570796, 1.853980],accel_mss,speed_ms,0,blend_radius_m)
    movel([0.286595, -1.337958, -2.600796, -0.773635, 1.570796, 1.857391],accel_mss,speed_ms,0,blend_radius_m)
    movel([0.287232, -1.337738, -2.600939, -0.773713, 1.570796, 1.858028],accel_mss,speed_ms,0,blend_radius_m)
    movel([0.287280, -1.337583, -2.601038, -0.773767, 1.570796, 1.858076],accel_mss,speed_ms,0,blend_radius_m)
    movel([0.287160, -1.337413, -2.601149, -0.773828, 1.570796, 1.857956],accel_mss,speed_ms,0,blend_radius_m)
    movel([0.287483, -1.335974, -2.602075, -0.774340, 1.570796, 1.858279],accel_mss,speed_ms,0,blend_radius_m)
    movel([0.288182, -1.333702, -2.603533, -0.775154, 1.570796, 1.858978],accel_mss,speed_ms,0,blend_radius_m)
    movel([0.289249, -1.330434, -2.605618, -0.776337, 1.570796, 1.860045],accel_mss,speed_ms,0,blend_radius_m)
    movel([0.289499, -1.329908, -2.605952, -0.776529, 1.570796, 1.860295],accel_mss,speed_ms,0,blend_radius_m)
    movel([0.289759, -1.329653, -2.606114, -0.776622, 1.570796, 1.860556],accel_mss,speed_ms,0,blend_radius_m)
    movel([0.290150, -1.329547, -2.606181, -0.776661, 1.570796, 1.860946],accel_mss,speed_ms,0,blend_radius_m)
    movel([0.290332, -1.329711, -2.606077, -0.776601, 1.570796, 1.861128],accel_mss,speed_ms,0,blend_radius_m)
    movel([0.290278, -1.330282, -2.605714, -0.776392, 1.570796, 1.861074],accel_mss,speed_ms,0,blend_radius_m)
    movel([0.289344, -1.333607, -2.603594, -0.775188, 1.570796, 1.860140],accel_mss,speed_ms,0,blend_radius_m)
    movel([0.290294, -1.332239, -2.604468, -0.775682, 1.570796, 1.861090],accel_mss,speed_ms,0,blend_radius_m)
    movel([0.291538, -1.330556, -2.605540, -0.776293, 1.570796, 1.862335],accel_mss,speed_ms,0,blend_radius_m)
    movel([0.293326, -1.328342, -2.606945, -0.777102, 1.570796, 1.864122],accel_mss,speed_ms,0,blend_radius_m)
    movel([0.297343, -1.323736, -2.609846, -0.778807, 1.570796, 1.868139],accel_mss,speed_ms,0,blend_radius_m)
    movel([0.299726, -1.321195, -2.611434, -0.779760, 1.570796, 1.870523],accel_mss,speed_ms,0,blend_radius_m)
    movel([0.305451, -1.315342, -2.615059, -0.781988, 1.570796, 1.876247],accel_mss,speed_ms,0,blend_radius_m)
    movel([0.306359, -1.314537, -2.615554, -0.782298, 1.570796, 1.877155],accel_mss,speed_ms,0,blend_radius_m)
    movel([0.306784, -1.314262, -2.615723, -0.782404, 1.570796, 1.877581],accel_mss,speed_ms,0,blend_radius_m)
    movel([0.307136, -1.314157, -2.615788, -0.782444, 1.570796, 1.877933],accel_mss,speed_ms,0,blend_radius_m)
    movel([0.307327, -1.314243, -2.615735, -0.782411, 1.570796, 1.878123],accel_mss,speed_ms,0,blend_radius_m)
    movel([0.307338, -1.314482, -2.615588, -0.782319, 1.570796, 1.878134],accel_mss,speed_ms,0,blend_radius_m)
    movel([0.307220, -1.314675, -2.615469, -0.782244, 1.570796, 1.878016],accel_mss,speed_ms,0,blend_radius_m)
    movel([0.306316, -1.315640, -2.614876, -0.781873, 1.570796, 1.877112],accel_mss,speed_ms,0,blend_radius_m)
    movel([0.299054, -1.323144, -2.610217, -0.779029, 1.570796, 1.869851],accel_mss,speed_ms,0,blend_radius_m)
    movel([0.296977, -1.325385, -2.608810, -0.778194, 1.570796, 1.867773],accel_mss,speed_ms,0,blend_radius_m)
    movel([0.294865, -1.327839, -2.607263, -0.777287, 1.570796, 1.865662],accel_mss,speed_ms,0,blend_radius_m)
    movel([0.296871, -1.326178, -2.608312, -0.777900, 1.570796, 1.867668],accel_mss,speed_ms,0,blend_radius_m)
    movel([0.298173, -1.325140, -2.608964, -0.778284, 1.570796, 1.868970],accel_mss,speed_ms,0,blend_radius_m)
    movel([0.299000, -1.324601, -2.609303, -0.778485, 1.570796, 1.869797],accel_mss,speed_ms,0,blend_radius_m)
    movel([0.299468, -1.324470, -2.609385, -0.778534, 1.570796, 1.870264],accel_mss,speed_ms,0,blend_radius_m)
    movel([0.299683, -1.324652, -2.609271, -0.778466, 1.570796, 1.870479],accel_mss,speed_ms,0,blend_radius_m)
    movel([0.299343, -1.325448, -2.608771, -0.778170, 1.570796, 1.870139],accel_mss,speed_ms,0,blend_radius_m)
    movel([0.298956, -1.326194, -2.608301, -0.777894, 1.570796, 1.869753],accel_mss,speed_ms,0,blend_radius_m)
    movel([0.297343, -1.329155, -2.606430, -0.776804, 1.570796, 1.868140],accel_mss,speed_ms,0,blend_radius_m)
    movel([0.297708, -1.329010, -2.606522, -0.776857, 1.570796, 1.868504],accel_mss,speed_ms,0,blend_radius_m)
    movel([0.298085, -1.328757, -2.606682, -0.776950, 1.570796, 1.868881],accel_mss,speed_ms,0,blend_radius_m)
    movel([0.301785, -1.326345, -2.608206, -0.777838, 1.570796, 1.872581],accel_mss,speed_ms,0,blend_radius_m)
    movel([0.303242, -1.325449, -2.608770, -0.778170, 1.570796, 1.874038],accel_mss,speed_ms,0,blend_radius_m)
    movel([0.307752, -1.322628, -2.610539, -0.779222, 1.570796, 1.878549],accel_mss,speed_ms,0,blend_radius_m)
    movel([0.309030, -1.321704, -2.611116, -0.779569, 1.570796, 1.879826],accel_mss,speed_ms,0,blend_radius_m)
    movel([0.311488, -1.319734, -2.612343, -0.780312, 1.570796, 1.882284],accel_mss,speed_ms,0,blend_radius_m)
    movel([0.312160, -1.319308, -2.612608, -0.780473, 1.570796, 1.882957],accel_mss,speed_ms,0,blend_radius_m)
    movel([0.312546, -1.319224, -2.612660, -0.780505, 1.570796, 1.883343],accel_mss,speed_ms,0,blend_radius_m)
    movel([0.312722, -1.319401, -2.612550, -0.780438, 1.570796, 1.883518],accel_mss,speed_ms,0,blend_radius_m)
    movel([0.312558, -1.319995, -2.612181, -0.780213, 1.570796, 1.883355],accel_mss,speed_ms,0,blend_radius_m)
    movel([0.311508, -1.321762, -2.611080, -0.779547, 1.570796, 1.882305],accel_mss,speed_ms,0,blend_radius_m)
    movel([0.310330, -1.323591, -2.609937, -0.778862, 1.570796, 1.881126],accel_mss,speed_ms,0,blend_radius_m)
    movel([0.309265, -1.325038, -2.609029, -0.778323, 1.570796, 1.880062],accel_mss,speed_ms,0,blend_radius_m)
    movel([0.308039, -1.326663, -2.608006, -0.777720, 1.570796, 1.878835],accel_mss,speed_ms,0,blend_radius_m)
    movel([0.308604, -1.326472, -2.608126, -0.777791, 1.570796, 1.879401],accel_mss,speed_ms,0,blend_radius_m)
    movel([0.311317, -1.324515, -2.609357, -0.778517, 1.570796, 1.882114],accel_mss,speed_ms,0,blend_radius_m)
    movel([0.316231, -1.320761, -2.611704, -0.779924, 1.570796, 1.887027],accel_mss,speed_ms,0,blend_radius_m)
    movel([0.319315, -1.318232, -2.613275, -0.780882, 1.570796, 1.890112],accel_mss,speed_ms,0,blend_radius_m)
    movel([0.321777, -1.313516, -2.616181, -0.782692, 1.570796, 1.892573],accel_mss,speed_ms,0,blend_radius_m)
    movel([0.322832, -1.311340, -2.617512, -0.783537, 1.570796, 1.893628],accel_mss,speed_ms,0,blend_radius_m)
    movel([0.325390, -1.305459, -2.621078, -0.785852, 1.570796, 1.896186],accel_mss,speed_ms,0,blend_radius_m)
    movel([0.325692, -1.304844, -2.621448, -0.786096, 1.570796, 1.896488],accel_mss,speed_ms,0,blend_radius_m)
    movel([0.325935, -1.304661, -2.621559, -0.786170, 1.570796, 1.896731],accel_mss,speed_ms,0,blend_radius_m)
    movel([0.326078, -1.304646, -2.621567, -0.786175, 1.570796, 1.896874],accel_mss,speed_ms,0,blend_radius_m)
    movel([0.326355, -1.304704, -2.621533, -0.786152, 1.570796, 1.897152],accel_mss,speed_ms,0,blend_radius_m)
    movel([0.326482, -1.304865, -2.621436, -0.786088, 1.570796, 1.897279],accel_mss,speed_ms,0,blend_radius_m)
    movel([0.326323, -1.305625, -2.620978, -0.785786, 1.570796, 1.897119],accel_mss,speed_ms,0,blend_radius_m)
    movel([0.325852, -1.306810, -2.620263, -0.785316, 1.570796, 1.896648],accel_mss,speed_ms,0,blend_radius_m)
    movel([0.324104, -1.310798, -2.617842, -0.783748, 1.570796, 1.894901],accel_mss,speed_ms,0,blend_radius_m)
    movel([0.321872, -1.315339, -2.615061, -0.781989, 1.570796, 1.892669],accel_mss,speed_ms,0,blend_radius_m)
    movel([0.319480, -1.319814, -2.612293, -0.780282, 1.570796, 1.890277],accel_mss,speed_ms,0,blend_radius_m)
    movel([0.317242, -1.323608, -2.609926, -0.778855, 1.570796, 1.888038],accel_mss,speed_ms,0,blend_radius_m)
    movel([0.317155, -1.323849, -2.609775, -0.778765, 1.570796, 1.887952],accel_mss,speed_ms,0,blend_radius_m)
    movel([0.317956, -1.323688, -2.609876, -0.778825, 1.570796, 1.888753],accel_mss,speed_ms,0,blend_radius_m)
    movel([0.318492, -1.323773, -2.609823, -0.778794, 1.570796, 1.889289],accel_mss,speed_ms,0,blend_radius_m)
    movel([0.318947, -1.324003, -2.609678, -0.778708, 1.570796, 1.889743],accel_mss,speed_ms,0,blend_radius_m)
    movel([0.319213, -1.324339, -2.609468, -0.778583, 1.570796, 1.890009],accel_mss,speed_ms,0,blend_radius_m)
    movel([0.319354, -1.325133, -2.608969, -0.778287, 1.570796, 1.890150],accel_mss,speed_ms,0,blend_radius_m)
    movel([0.319202, -1.326139, -2.608336, -0.777914, 1.570796, 1.889999],accel_mss,speed_ms,0,blend_radius_m)
    movel([0.318708, -1.327569, -2.607434, -0.777386, 1.570796, 1.889504],accel_mss,speed_ms,0,blend_radius_m)
    movel([0.317731, -1.329792, -2.606026, -0.776571, 1.570796, 1.888527],accel_mss,speed_ms,0,blend_radius_m)
    movel([0.316211, -1.333385, -2.603736, -0.775268, 1.570796, 1.887007],accel_mss,speed_ms,0,blend_radius_m)
    movel([0.315417, -1.335514, -2.602371, -0.774504, 1.570796, 1.886213],accel_mss,speed_ms,0,blend_radius_m)
    movel([0.312480, -1.343953, -2.596900, -0.771537, 1.570796, 1.883276],accel_mss,speed_ms,0,blend_radius_m)
    movel([0.312677, -1.345001, -2.596213, -0.771175, 1.570796, 1.883474],accel_mss,speed_ms,0,blend_radius_m)
    movel([0.313283, -1.346907, -2.594961, -0.770521, 1.570796, 1.884079],accel_mss,speed_ms,0,blend_radius_m)
    movel([0.314864, -1.350096, -2.592855, -0.769438, 1.570796, 1.885661],accel_mss,speed_ms,0,blend_radius_m)
    movel([0.316580, -1.353176, -2.590808, -0.768405, 1.570796, 1.887376],accel_mss,speed_ms,0,blend_radius_m)
    movel([0.317108, -1.353941, -2.590297, -0.768151, 1.570796, 1.887904],accel_mss,speed_ms,0,blend_radius_m)
    movel([0.318419, -1.355167, -2.589477, -0.767745, 1.570796, 1.889215],accel_mss,speed_ms,0,blend_radius_m)
    movel([0.319308, -1.355696, -2.589123, -0.767570, 1.570796, 1.890104],accel_mss,speed_ms,0,blend_radius_m)
    movel([0.320203, -1.356143, -2.588823, -0.767423, 1.570796, 1.890999],accel_mss,speed_ms,0,blend_radius_m)
    movel([0.320483, -1.356076, -2.588868, -0.767445, 1.570796, 1.891279],accel_mss,speed_ms,0,blend_radius_m)
    movel([0.320592, -1.355849, -2.589020, -0.767520, 1.570796, 1.891388],accel_mss,speed_ms,0,blend_radius_m)
    movel([0.320419, -1.355300, -2.589388, -0.767701, 1.570796, 1.891215],accel_mss,speed_ms,0,blend_radius_m)
    movel([0.318422, -1.351419, -2.591977, -0.768993, 1.570796, 1.889218],accel_mss,speed_ms,0,blend_radius_m)
    movel([0.317671, -1.349417, -2.593305, -0.769667, 1.570796, 1.888467],accel_mss,speed_ms,0,blend_radius_m)
    movel([0.317183, -1.347311, -2.594695, -0.770383, 1.570796, 1.887979],accel_mss,speed_ms,0,blend_radius_m)
    movel([0.316915, -1.344971, -2.596233, -0.771185, 1.570796, 1.887711],accel_mss,speed_ms,0,blend_radius_m)
    movel([0.316884, -1.343933, -2.596913, -0.771544, 1.570796, 1.887681],accel_mss,speed_ms,0,blend_radius_m)
    movel([0.316976, -1.343284, -2.597337, -0.771768, 1.570796, 1.887772],accel_mss,speed_ms,0,blend_radius_m)
    movel([0.317192, -1.342911, -2.597580, -0.771897, 1.570796, 1.887988],accel_mss,speed_ms,0,blend_radius_m)
    movel([0.317521, -1.342732, -2.597697, -0.771960, 1.570796, 1.888317],accel_mss,speed_ms,0,blend_radius_m)
    movel([0.317882, -1.342894, -2.597591, -0.771903, 1.570796, 1.888678],accel_mss,speed_ms,0,blend_radius_m)
    movel([0.317971, -1.343211, -2.597384, -0.771793, 1.570796, 1.888767],accel_mss,speed_ms,0,blend_radius_m)
    movel([0.318218, -1.344826, -2.596328, -0.771235, 1.570796, 1.889015],accel_mss,speed_ms,0,blend_radius_m)
    movel([0.318473, -1.345681, -2.595767, -0.770941, 1.570796, 1.889269],accel_mss,speed_ms,0,blend_radius_m)
    movel([0.318755, -1.346389, -2.595302, -0.770698, 1.570796, 1.889552],accel_mss,speed_ms,0,blend_radius_m)
    movel([0.318911, -1.346354, -2.595325, -0.770710, 1.570796, 1.889708],accel_mss,speed_ms,0,blend_radius_m)
    movel([0.319055, -1.345936, -2.595600, -0.770853, 1.570796, 1.889851],accel_mss,speed_ms,0,blend_radius_m)
    movel([0.319027, -1.344683, -2.596422, -0.771284, 1.570796, 1.889823],accel_mss,speed_ms,0,blend_radius_m)
    movel([0.318491, -1.339562, -2.599759, -0.773069, 1.570796, 1.889288],accel_mss,speed_ms,0,blend_radius_m)
    movel([0.318600, -1.337704, -2.600961, -0.773725, 1.570796, 1.889396],accel_mss,speed_ms,0,blend_radius_m)
    movel([0.318976, -1.336335, -2.601843, -0.774211, 1.570796, 1.889772],accel_mss,speed_ms,0,blend_radius_m)
    movel([0.319226, -1.335994, -2.602062, -0.774332, 1.570796, 1.890023],accel_mss,speed_ms,0,blend_radius_m)
    movel([0.319605, -1.335796, -2.602190, -0.774403, 1.570796, 1.890401],accel_mss,speed_ms,0,blend_radius_m)
    movel([0.319854, -1.335797, -2.602189, -0.774403, 1.570796, 1.890650],accel_mss,speed_ms,0,blend_radius_m)
    movel([0.319963, -1.335932, -2.602102, -0.774355, 1.570796, 1.890759],accel_mss,speed_ms,0,blend_radius_m)
    movel([0.319945, -1.336287, -2.601874, -0.774228, 1.570796, 1.890741],accel_mss,speed_ms,0,blend_radius_m)
    movel([0.319589, -1.338312, -2.600568, -0.773509, 1.570796, 1.890386],accel_mss,speed_ms,0,blend_radius_m)
    movel([0.319629, -1.338970, -2.600142, -0.773277, 1.570796, 1.890426],accel_mss,speed_ms,0,blend_radius_m)
    movel([0.319894, -1.339507, -2.599794, -0.773088, 1.570796, 1.890691],accel_mss,speed_ms,0,blend_radius_m)
    movel([0.320502, -1.340161, -2.599370, -0.772858, 1.570796, 1.891299],accel_mss,speed_ms,0,blend_radius_m)
    movel([0.321881, -1.341917, -2.598229, -0.772244, 1.570796, 1.892677],accel_mss,speed_ms,0,blend_radius_m)
    movel([0.322256, -1.342558, -2.597811, -0.772020, 1.570796, 1.893053],accel_mss,speed_ms,0,blend_radius_m)
    movel([0.323168, -1.343959, -2.596896, -0.771534, 1.570796, 1.893964],accel_mss,speed_ms,0,blend_radius_m)
    movel([0.323281, -1.343973, -2.596887, -0.771530, 1.570796, 1.894077],accel_mss,speed_ms,0,blend_radius_m)
    movel([0.323513, -1.343747, -2.597034, -0.771608, 1.570796, 1.894309],accel_mss,speed_ms,0,blend_radius_m)
    movel([0.323658, -1.343241, -2.597365, -0.771783, 1.570796, 1.894454],accel_mss,speed_ms,0,blend_radius_m)
    movel([0.323698, -1.342643, -2.597755, -0.771991, 1.570796, 1.894494],accel_mss,speed_ms,0,blend_radius_m)
    movel([0.323602, -1.342093, -2.598114, -0.772182, 1.570796, 1.894399],accel_mss,speed_ms,0,blend_radius_m)
    movel([0.321867, -1.337613, -2.601019, -0.773757, 1.570796, 1.892663],accel_mss,speed_ms,0,blend_radius_m)
    movel([0.321389, -1.335317, -2.602497, -0.774574, 1.570796, 1.892185],accel_mss,speed_ms,0,blend_radius_m)
    movel([0.321267, -1.332851, -2.604077, -0.775460, 1.570796, 1.892063],accel_mss,speed_ms,0,blend_radius_m)
    movel([0.321484, -1.330010, -2.605887, -0.776492, 1.570796, 1.892280],accel_mss,speed_ms,0,blend_radius_m)
    movel([0.321947, -1.325584, -2.608685, -0.778120, 1.570796, 1.892744],accel_mss,speed_ms,0,blend_radius_m)
    movel([0.322151, -1.324985, -2.609062, -0.778342, 1.570796, 1.892947],accel_mss,speed_ms,0,blend_radius_m)
    movel([0.322456, -1.324610, -2.609297, -0.778481, 1.570796, 1.893253],accel_mss,speed_ms,0,blend_radius_m)
    movel([0.322846, -1.324433, -2.609408, -0.778547, 1.570796, 1.893642],accel_mss,speed_ms,0,blend_radius_m)
    movel([0.323256, -1.324559, -2.609330, -0.778501, 1.570796, 1.894053],accel_mss,speed_ms,0,blend_radius_m)
    movel([0.323504, -1.324700, -2.609241, -0.778448, 1.570796, 1.894301],accel_mss,speed_ms,0,blend_radius_m)
    movel([0.323712, -1.324524, -2.609351, -0.778513, 1.570796, 1.894508],accel_mss,speed_ms,0,blend_radius_m)
    movel([0.324194, -1.322274, -2.610760, -0.779354, 1.570796, 1.894991],accel_mss,speed_ms,0,blend_radius_m)
    movel([0.324385, -1.320762, -2.611704, -0.779923, 1.570796, 1.895181],accel_mss,speed_ms,0,blend_radius_m)
    movel([0.324865, -1.317732, -2.613584, -0.781073, 1.570796, 1.895661],accel_mss,speed_ms,0,blend_radius_m)
    movel([0.325178, -1.316424, -2.614392, -0.781573, 1.570796, 1.895975],accel_mss,speed_ms,0,blend_radius_m)
    movel([0.325480, -1.315651, -2.614869, -0.781869, 1.570796, 1.896276],accel_mss,speed_ms,0,blend_radius_m)
    movel([0.325973, -1.314833, -2.615372, -0.782184, 1.570796, 1.896770],accel_mss,speed_ms,0,blend_radius_m)
    movel([0.326495, -1.314300, -2.615700, -0.782389, 1.570796, 1.897291],accel_mss,speed_ms,0,blend_radius_m)
    movel([0.327012, -1.314074, -2.615839, -0.782477, 1.570796, 1.897808],accel_mss,speed_ms,0,blend_radius_m)
    movel([0.327771, -1.314220, -2.615749, -0.782420, 1.570796, 1.898568],accel_mss,speed_ms,0,blend_radius_m)
    movel([0.327825, -1.310294, -2.618149, -0.783945, 1.570796, 1.898621],accel_mss,speed_ms,0,blend_radius_m)
    movel([0.328013, -1.308741, -2.619093, -0.784554, 1.570796, 1.898810],accel_mss,speed_ms,0,blend_radius_m)
    movel([0.328332, -1.307287, -2.619975, -0.785128, 1.570796, 1.899128],accel_mss,speed_ms,0,blend_radius_m)
    movel([0.328796, -1.305856, -2.620839, -0.785694, 1.570796, 1.899592],accel_mss,speed_ms,0,blend_radius_m)
    movel([0.329396, -1.304434, -2.621695, -0.786260, 1.570796, 1.900192],accel_mss,speed_ms,0,blend_radius_m)
    movel([0.329591, -1.304261, -2.621799, -0.786329, 1.570796, 1.900387],accel_mss,speed_ms,0,blend_radius_m)
    movel([0.330132, -1.304196, -2.621838, -0.786355, 1.570796, 1.900928],accel_mss,speed_ms,0,blend_radius_m)
    movel([0.330220, -1.304331, -2.621757, -0.786301, 1.570796, 1.901016],accel_mss,speed_ms,0,blend_radius_m)
    movel([0.329395, -1.307235, -2.620006, -0.785148, 1.570796, 1.900191],accel_mss,speed_ms,0,blend_radius_m)
    movel([0.329118, -1.308609, -2.619174, -0.784606, 1.570796, 1.899914],accel_mss,speed_ms,0,blend_radius_m)
    movel([0.328917, -1.311912, -2.617163, -0.783314, 1.570796, 1.899714],accel_mss,speed_ms,0,blend_radius_m)
    movel([0.328897, -1.313456, -2.616218, -0.782715, 1.570796, 1.899694],accel_mss,speed_ms,0,blend_radius_m)
    movel([0.328838, -1.314044, -2.615857, -0.782488, 1.570796, 1.899634],accel_mss,speed_ms,0,blend_radius_m)
    movel([0.328695, -1.314426, -2.615622, -0.782341, 1.570796, 1.899491],accel_mss,speed_ms,0,blend_radius_m)
    movel([0.328122, -1.315083, -2.615218, -0.782087, 1.570796, 1.898918],accel_mss,speed_ms,0,blend_radius_m)
    movel([0.327900, -1.315229, -2.615129, -0.782031, 1.570796, 1.898697],accel_mss,speed_ms,0,blend_radius_m)
    movel([0.327015, -1.315300, -2.615085, -0.782004, 1.570796, 1.897811],accel_mss,speed_ms,0,blend_radius_m)
    movel([0.326814, -1.315349, -2.615055, -0.781985, 1.570796, 1.897611],accel_mss,speed_ms,0,blend_radius_m)
    movel([0.326505, -1.315650, -2.614869, -0.781869, 1.570796, 1.897301],accel_mss,speed_ms,0,blend_radius_m)
    movel([0.326243, -1.316211, -2.614524, -0.781654, 1.570796, 1.897040],accel_mss,speed_ms,0,blend_radius_m)
    movel([0.325771, -1.318529, -2.613091, -0.780769, 1.570796, 1.896567],accel_mss,speed_ms,0,blend_radius_m)
    movel([0.325555, -1.320254, -2.612020, -0.780115, 1.570796, 1.896352],accel_mss,speed_ms,0,blend_radius_m)
    movel([0.325022, -1.323589, -2.609938, -0.778862, 1.570796, 1.895818],accel_mss,speed_ms,0,blend_radius_m)
    movel([0.324690, -1.324561, -2.609328, -0.778500, 1.570796, 1.895486],accel_mss,speed_ms,0,blend_radius_m)
    movel([0.324022, -1.325521, -2.608725, -0.778143, 1.570796, 1.894818],accel_mss,speed_ms,0,blend_radius_m)
    movel([0.323792, -1.325718, -2.608601, -0.778070, 1.570796, 1.894589],accel_mss,speed_ms,0,blend_radius_m)
    movel([0.323215, -1.325936, -2.608463, -0.777989, 1.570796, 1.894011],accel_mss,speed_ms,0,blend_radius_m)
    movel([0.323016, -1.326320, -2.608222, -0.777847, 1.570796, 1.893813],accel_mss,speed_ms,0,blend_radius_m)
    movel([0.322996, -1.326543, -2.608081, -0.777765, 1.570796, 1.893792],accel_mss,speed_ms,0,blend_radius_m)
    movel([0.322922, -1.327522, -2.607463, -0.777404, 1.570796, 1.893719],accel_mss,speed_ms,0,blend_radius_m)
    movel([0.323757, -1.327313, -2.607595, -0.777481, 1.570796, 1.894554],accel_mss,speed_ms,0,blend_radius_m)
    movel([0.324353, -1.327267, -2.607625, -0.777498, 1.570796, 1.895149],accel_mss,speed_ms,0,blend_radius_m)
    movel([0.324871, -1.327374, -2.607557, -0.777458, 1.570796, 1.895667],accel_mss,speed_ms,0,blend_radius_m)
    movel([0.325226, -1.327625, -2.607398, -0.777366, 1.570796, 1.896022],accel_mss,speed_ms,0,blend_radius_m)
    movel([0.325575, -1.328047, -2.607131, -0.777210, 1.570796, 1.896372],accel_mss,speed_ms,0,blend_radius_m)
    movel([0.326235, -1.326974, -2.607809, -0.777606, 1.570796, 1.897031],accel_mss,speed_ms,0,blend_radius_m)
    movel([0.328106, -1.323722, -2.609854, -0.778813, 1.570796, 1.898903],accel_mss,speed_ms,0,blend_radius_m)
    movel([0.328918, -1.322139, -2.610845, -0.779405, 1.570796, 1.899714],accel_mss,speed_ms,0,blend_radius_m)
    movel([0.330408, -1.318912, -2.612853, -0.780624, 1.570796, 1.901205],accel_mss,speed_ms,0,blend_radius_m)
    movel([0.330828, -1.318132, -2.613337, -0.780920, 1.570796, 1.901624],accel_mss,speed_ms,0,blend_radius_m)
    movel([0.331157, -1.317737, -2.613581, -0.781071, 1.570796, 1.901953],accel_mss,speed_ms,0,blend_radius_m)
    movel([0.331497, -1.317570, -2.613685, -0.781135, 1.570796, 1.902293],accel_mss,speed_ms,0,blend_radius_m)
    movel([0.331716, -1.317732, -2.613584, -0.781073, 1.570796, 1.902512],accel_mss,speed_ms,0,blend_radius_m)
    movel([0.331642, -1.318314, -2.613224, -0.780851, 1.570796, 1.902438],accel_mss,speed_ms,0,blend_radius_m)
    movel([0.330607, -1.320847, -2.611650, -0.779891, 1.570796, 1.901404],accel_mss,speed_ms,0,blend_radius_m)
    movel([0.329166, -1.323665, -2.609890, -0.778834, 1.570796, 1.899962],accel_mss,speed_ms,0,blend_radius_m)
    movel([0.327273, -1.326926, -2.607839, -0.777623, 1.570796, 1.898070],accel_mss,speed_ms,0,blend_radius_m)
    movel([0.325373, -1.329976, -2.605909, -0.776504, 1.570796, 1.896170],accel_mss,speed_ms,0,blend_radius_m)
    movel([0.325015, -1.330423, -2.605625, -0.776341, 1.570796, 1.895812],accel_mss,speed_ms,0,blend_radius_m)
    movel([0.324562, -1.330803, -2.605383, -0.776203, 1.570796, 1.895358],accel_mss,speed_ms,0,blend_radius_m)
    movel([0.324167, -1.330987, -2.605266, -0.776136, 1.570796, 1.894963],accel_mss,speed_ms,0,blend_radius_m)
    movel([0.323949, -1.330918, -2.605310, -0.776161, 1.570796, 1.894746],accel_mss,speed_ms,0,blend_radius_m)
    movel([0.323927, -1.330567, -2.605534, -0.776289, 1.570796, 1.894724],accel_mss,speed_ms,0,blend_radius_m)
    movel([0.324129, -1.329871, -2.605976, -0.776542, 1.570796, 1.894926],accel_mss,speed_ms,0,blend_radius_m)
    movel([0.324363, -1.328987, -2.606536, -0.776866, 1.570796, 1.895159],accel_mss,speed_ms,0,blend_radius_m)
    movel([0.324344, -1.328731, -2.606699, -0.776960, 1.570796, 1.895140],accel_mss,speed_ms,0,blend_radius_m)
    movel([0.324031, -1.328317, -2.606961, -0.777111, 1.570796, 1.894827],accel_mss,speed_ms,0,blend_radius_m)
    movel([0.323801, -1.328255, -2.607000, -0.777134, 1.570796, 1.894597],accel_mss,speed_ms,0,blend_radius_m)
    movel([0.323131, -1.328553, -2.606811, -0.777025, 1.570796, 1.893927],accel_mss,speed_ms,0,blend_radius_m)
    movel([0.322888, -1.328760, -2.606680, -0.776949, 1.570796, 1.893685],accel_mss,speed_ms,0,blend_radius_m)
    movel([0.322657, -1.329318, -2.606326, -0.776744, 1.570796, 1.893453],accel_mss,speed_ms,0,blend_radius_m)
    movel([0.322539, -1.330121, -2.605817, -0.776451, 1.570796, 1.893335],accel_mss,speed_ms,0,blend_radius_m)
    movel([0.322382, -1.332635, -2.604215, -0.775539, 1.570796, 1.893178],accel_mss,speed_ms,0,blend_radius_m)
    movel([0.322593, -1.335105, -2.602633, -0.774650, 1.570796, 1.893389],accel_mss,speed_ms,0,blend_radius_m)
    movel([0.323175, -1.337561, -2.601053, -0.773775, 1.570796, 1.893971],accel_mss,speed_ms,0,blend_radius_m)
    movel([0.324127, -1.340038, -2.599450, -0.772901, 1.570796, 1.894923],accel_mss,speed_ms,0,blend_radius_m)
    movel([0.324561, -1.341118, -2.598749, -0.772523, 1.570796, 1.895357],accel_mss,speed_ms,0,blend_radius_m)
    movel([0.324768, -1.341983, -2.598186, -0.772221, 1.570796, 1.895564],accel_mss,speed_ms,0,blend_radius_m)
    movel([0.324777, -1.342755, -2.597682, -0.771952, 1.570796, 1.895574],accel_mss,speed_ms,0,blend_radius_m)
    movel([0.324601, -1.343530, -2.597176, -0.771683, 1.570796, 1.895397],accel_mss,speed_ms,0,blend_radius_m)
    movel([0.324257, -1.344260, -2.596699, -0.771430, 1.570796, 1.895054],accel_mss,speed_ms,0,blend_radius_m)
    movel([0.324034, -1.344507, -2.596537, -0.771345, 1.570796, 1.894831],accel_mss,speed_ms,0,blend_radius_m)
    movel([0.323141, -1.345079, -2.596162, -0.771148, 1.570796, 1.893937],accel_mss,speed_ms,0,blend_radius_m)
    movel([0.322703, -1.345110, -2.596142, -0.771137, 1.570796, 1.893499],accel_mss,speed_ms,0,blend_radius_m)
    movel([0.322296, -1.344845, -2.596316, -0.771229, 1.570796, 1.893092],accel_mss,speed_ms,0,blend_radius_m)
    movel([0.321779, -1.344151, -2.596770, -0.771468, 1.570796, 1.892576],accel_mss,speed_ms,0,blend_radius_m)
    movel([0.319826, -1.341322, -2.598616, -0.772451, 1.570796, 1.890622],accel_mss,speed_ms,0,blend_radius_m)
    movel([0.320027, -1.342711, -2.597711, -0.771967, 1.570796, 1.890824],accel_mss,speed_ms,0,blend_radius_m)
    movel([0.320162, -1.345078, -2.596163, -0.771148, 1.570796, 1.890958],accel_mss,speed_ms,0,blend_radius_m)
    movel([0.320058, -1.346013, -2.595549, -0.770827, 1.570796, 1.890854],accel_mss,speed_ms,0,blend_radius_m)
    movel([0.319830, -1.346613, -2.595155, -0.770621, 1.570796, 1.890626],accel_mss,speed_ms,0,blend_radius_m)
    movel([0.319671, -1.346830, -2.595012, -0.770547, 1.570796, 1.890467],accel_mss,speed_ms,0,blend_radius_m)
    movel([0.319236, -1.347196, -2.594771, -0.770422, 1.570796, 1.890032],accel_mss,speed_ms,0,blend_radius_m)
    movel([0.318973, -1.347327, -2.594685, -0.770377, 1.570796, 1.889769],accel_mss,speed_ms,0,blend_radius_m)
    movel([0.318397, -1.347567, -2.594526, -0.770296, 1.570796, 1.889193],accel_mss,speed_ms,0,blend_radius_m)
    movel([0.318594, -1.348296, -2.594046, -0.770047, 1.570796, 1.889390],accel_mss,speed_ms,0,blend_radius_m)
    movel([0.319373, -1.350480, -2.592600, -0.769308, 1.570796, 1.890169],accel_mss,speed_ms,0,blend_radius_m)
    movel([0.319914, -1.351632, -2.591836, -0.768921, 1.570796, 1.890710],accel_mss,speed_ms,0,blend_radius_m)
    movel([0.321313, -1.354242, -2.590096, -0.768051, 1.570796, 1.892110],accel_mss,speed_ms,0,blend_radius_m)
    movel([0.321691, -1.355242, -2.589427, -0.767720, 1.570796, 1.892488],accel_mss,speed_ms,0,blend_radius_m)
    movel([0.321788, -1.356029, -2.588899, -0.767461, 1.570796, 1.892584],accel_mss,speed_ms,0,blend_radius_m)
    movel([0.321625, -1.356737, -2.588424, -0.767228, 1.570796, 1.892421],accel_mss,speed_ms,0,blend_radius_m)
    movel([0.321353, -1.357027, -2.588229, -0.767133, 1.570796, 1.892150],accel_mss,speed_ms,0,blend_radius_m)
    movel([0.321111, -1.357096, -2.588183, -0.767110, 1.570796, 1.891907],accel_mss,speed_ms,0,blend_radius_m)
    movel([0.320654, -1.357148, -2.588148, -0.767093, 1.570796, 1.891451],accel_mss,speed_ms,0,blend_radius_m)
    movel([0.319732, -1.357074, -2.588198, -0.767118, 1.570796, 1.890528],accel_mss,speed_ms,0,blend_radius_m)
    movel([0.319205, -1.356915, -2.588304, -0.767170, 1.570796, 1.890001],accel_mss,speed_ms,0,blend_radius_m)
    movel([0.318602, -1.356635, -2.588492, -0.767261, 1.570796, 1.889398],accel_mss,speed_ms,0,blend_radius_m)
    speed_ms = 0.005
    movel([0.318602, -1.347774, -2.584387, -0.780228, 1.570796, 1.889398],accel_mss,speed_ms,0,blend_radius_m)
    speed_ms = 0.040
    movel([0.352216, -1.331525, -2.594978, -0.785886, 1.570796, 1.923012],accel_mss,speed_ms,0,blend_radius_m)
    speed_ms = 0.005
    movel([0.352216, -1.340492, -2.599155, -0.772742, 1.570796, 1.923012],accel_mss,speed_ms,0,blend_radius_m)
    speed_ms = 0.025
    movel([0.352535, -1.340162, -2.599370, -0.772858, 1.570796, 1.923331],accel_mss,speed_ms,0,blend_radius_m)
    movel([0.352711, -1.339788, -2.599612, -0.772989, 1.570796, 1.923508],accel_mss,speed_ms,0,blend_radius_m)
    movel([0.352670, -1.338983, -2.600134, -0.773272, 1.570796, 1.923466],accel_mss,speed_ms,0,blend_radius_m)
    movel([0.352060, -1.338219, -2.600628, -0.773542, 1.570796, 1.922857],accel_mss,speed_ms,0,blend_radius_m)
    movel([0.350113, -1.337305, -2.601218, -0.773866, 1.570796, 1.920909],accel_mss,speed_ms,0,blend_radius_m)
    movel([0.349631, -1.337070, -2.601370, -0.773950, 1.570796, 1.920427],accel_mss,speed_ms,0,blend_radius_m)
    movel([0.348525, -1.336355, -2.601830, -0.774204, 1.570796, 1.919321],accel_mss,speed_ms,0,blend_radius_m)
    movel([0.348544, -1.336200, -2.601930, -0.774259, 1.570796, 1.919340],accel_mss,speed_ms,0,blend_radius_m)
    movel([0.348723, -1.335998, -2.602060, -0.774331, 1.570796, 1.919519],accel_mss,speed_ms,0,blend_radius_m)
    movel([0.349202, -1.335424, -2.602429, -0.774536, 1.570796, 1.919999],accel_mss,speed_ms,0,blend_radius_m)
    movel([0.349429, -1.334745, -2.602865, -0.774779, 1.570796, 1.920225],accel_mss,speed_ms,0,blend_radius_m)
    movel([0.349373, -1.333996, -2.603345, -0.775048, 1.570796, 1.920170],accel_mss,speed_ms,0,blend_radius_m)
    movel([0.349033, -1.333229, -2.603836, -0.775324, 1.570796, 1.919829],accel_mss,speed_ms,0,blend_radius_m)
    movel([0.348772, -1.332802, -2.604109, -0.775478, 1.570796, 1.919569],accel_mss,speed_ms,0,blend_radius_m)
    movel([0.351020, -1.333036, -2.603959, -0.775394, 1.570796, 1.921816],accel_mss,speed_ms,0,blend_radius_m)
    movel([0.352148, -1.332847, -2.604080, -0.775462, 1.570796, 1.922944],accel_mss,speed_ms,0,blend_radius_m)
    movel([0.353006, -1.332440, -2.604340, -0.775609, 1.570796, 1.923803],accel_mss,speed_ms,0,blend_radius_m)
    movel([0.353294, -1.332184, -2.604503, -0.775702, 1.570796, 1.924091],accel_mss,speed_ms,0,blend_radius_m)
    movel([0.353476, -1.331881, -2.604696, -0.775811, 1.570796, 1.924272],accel_mss,speed_ms,0,blend_radius_m)
    movel([0.353484, -1.331394, -2.605007, -0.775988, 1.570796, 1.924280],accel_mss,speed_ms,0,blend_radius_m)
    movel([0.353063, -1.330691, -2.605454, -0.776243, 1.570796, 1.923859],accel_mss,speed_ms,0,blend_radius_m)
    movel([0.352318, -1.329826, -2.606004, -0.776559, 1.570796, 1.923114],accel_mss,speed_ms,0,blend_radius_m)
    movel([0.349360, -1.326992, -2.607798, -0.777599, 1.570796, 1.920156],accel_mss,speed_ms,0,blend_radius_m)
    movel([0.348039, -1.325330, -2.608845, -0.778214, 1.570796, 1.918835],accel_mss,speed_ms,0,blend_radius_m)
    movel([0.347096, -1.323607, -2.609926, -0.778855, 1.570796, 1.917893],accel_mss,speed_ms,0,blend_radius_m)
    movel([0.346441, -1.321670, -2.611137, -0.779581, 1.570796, 1.917237],accel_mss,speed_ms,0,blend_radius_m)
    movel([0.346245, -1.320593, -2.611809, -0.779987, 1.570796, 1.917041],accel_mss,speed_ms,0,blend_radius_m)
    movel([0.346351, -1.320363, -2.611952, -0.780074, 1.570796, 1.917148],accel_mss,speed_ms,0,blend_radius_m)
    movel([0.347079, -1.319539, -2.612464, -0.780386, 1.570796, 1.917875],accel_mss,speed_ms,0,blend_radius_m)
    movel([0.347272, -1.319149, -2.612706, -0.780534, 1.570796, 1.918068],accel_mss,speed_ms,0,blend_radius_m)
    movel([0.347772, -1.317500, -2.613728, -0.781161, 1.570796, 1.918569],accel_mss,speed_ms,0,blend_radius_m)
    movel([0.347867, -1.316445, -2.614380, -0.781565, 1.570796, 1.918664],accel_mss,speed_ms,0,blend_radius_m)
    movel([0.347787, -1.315072, -2.615225, -0.782092, 1.570796, 1.918584],accel_mss,speed_ms,0,blend_radius_m)
    movel([0.347480, -1.312752, -2.616649, -0.782988, 1.570796, 1.918276],accel_mss,speed_ms,0,blend_radius_m)
    movel([0.347187, -1.309783, -2.618461, -0.784146, 1.570796, 1.917983],accel_mss,speed_ms,0,blend_radius_m)
    movel([0.347293, -1.309650, -2.618541, -0.784198, 1.570796, 1.918089],accel_mss,speed_ms,0,blend_radius_m)
    movel([0.348087, -1.309178, -2.618828, -0.784383, 1.570796, 1.918883],accel_mss,speed_ms,0,blend_radius_m)
    movel([0.348484, -1.308820, -2.619046, -0.784523, 1.570796, 1.919280],accel_mss,speed_ms,0,blend_radius_m)
    movel([0.348755, -1.308393, -2.619305, -0.784691, 1.570796, 1.919552],accel_mss,speed_ms,0,blend_radius_m)
    movel([0.349034, -1.307290, -2.619973, -0.785126, 1.570796, 1.919830],accel_mss,speed_ms,0,blend_radius_m)
    movel([0.348922, -1.305737, -2.620911, -0.785741, 1.570796, 1.919718],accel_mss,speed_ms,0,blend_radius_m)
    movel([0.348361, -1.303474, -2.622272, -0.786643, 1.570796, 1.919158],accel_mss,speed_ms,0,blend_radius_m)
    movel([0.348152, -1.302515, -2.622846, -0.787027, 1.570796, 1.918949],accel_mss,speed_ms,0,blend_radius_m)
    movel([0.348259, -1.302346, -2.622947, -0.787095, 1.570796, 1.919056],accel_mss,speed_ms,0,blend_radius_m)
    movel([0.349040, -1.301826, -2.623258, -0.787304, 1.570796, 1.919837],accel_mss,speed_ms,0,blend_radius_m)
    movel([0.349455, -1.301370, -2.623531, -0.787488, 1.570796, 1.920252],accel_mss,speed_ms,0,blend_radius_m)
    movel([0.350286, -1.299922, -2.624395, -0.788073, 1.570796, 1.921082],accel_mss,speed_ms,0,blend_radius_m)
    movel([0.350835, -1.298250, -2.625388, -0.788751, 1.570796, 1.921631],accel_mss,speed_ms,0,blend_radius_m)
    movel([0.350935, -1.296750, -2.626277, -0.789363, 1.570796, 1.921731],accel_mss,speed_ms,0,blend_radius_m)
    movel([0.350843, -1.295802, -2.626836, -0.789751, 1.570796, 1.921639],accel_mss,speed_ms,0,blend_radius_m)
    movel([0.351479, -1.295617, -2.626945, -0.789826, 1.570796, 1.922276],accel_mss,speed_ms,0,blend_radius_m)
    movel([0.352236, -1.295334, -2.627112, -0.789943, 1.570796, 1.923032],accel_mss,speed_ms,0,blend_radius_m)
    movel([0.352990, -1.294915, -2.627359, -0.790115, 1.570796, 1.923786],accel_mss,speed_ms,0,blend_radius_m)
    movel([0.353657, -1.294419, -2.627651, -0.790319, 1.570796, 1.924453],accel_mss,speed_ms,0,blend_radius_m)
    movel([0.354143, -1.293903, -2.627954, -0.790531, 1.570796, 1.924939],accel_mss,speed_ms,0,blend_radius_m)
    movel([0.354670, -1.293013, -2.628477, -0.790899, 1.570796, 1.925466],accel_mss,speed_ms,0,blend_radius_m)
    movel([0.355323, -1.291381, -2.629432, -0.791576, 1.570796, 1.926119],accel_mss,speed_ms,0,blend_radius_m)
    movel([0.355911, -1.289627, -2.630455, -0.792307, 1.570796, 1.926707],accel_mss,speed_ms,0,blend_radius_m)
    movel([0.356361, -1.287513, -2.631683, -0.793193, 1.570796, 1.927157],accel_mss,speed_ms,0,blend_radius_m)
    movel([0.356429, -1.286728, -2.632138, -0.793524, 1.570796, 1.927226],accel_mss,speed_ms,0,blend_radius_m)
    movel([0.356467, -1.284071, -2.633670, -0.794648, 1.570796, 1.927263],accel_mss,speed_ms,0,blend_radius_m)
    movel([0.356530, -1.283763, -2.633847, -0.794779, 1.570796, 1.927327],accel_mss,speed_ms,0,blend_radius_m)
    movel([0.356795, -1.283634, -2.633921, -0.794834, 1.570796, 1.927591],accel_mss,speed_ms,0,blend_radius_m)
    movel([0.357859, -1.283888, -2.633775, -0.794726, 1.570796, 1.928655],accel_mss,speed_ms,0,blend_radius_m)
    movel([0.358814, -1.284207, -2.633592, -0.794590, 1.570796, 1.929610],accel_mss,speed_ms,0,blend_radius_m)
    movel([0.357559, -1.284590, -2.633371, -0.794428, 1.570796, 1.928356],accel_mss,speed_ms,0,blend_radius_m)
    movel([0.357253, -1.284907, -2.633189, -0.794294, 1.570796, 1.928050],accel_mss,speed_ms,0,blend_radius_m)
    movel([0.357274, -1.285213, -2.633012, -0.794164, 1.570796, 1.928070],accel_mss,speed_ms,0,blend_radius_m)
    movel([0.357640, -1.285404, -2.632902, -0.794083, 1.570796, 1.928437],accel_mss,speed_ms,0,blend_radius_m)
    movel([0.359016, -1.285899, -2.632617, -0.793874, 1.570796, 1.929813],accel_mss,speed_ms,0,blend_radius_m)
    movel([0.359442, -1.286248, -2.632415, -0.793726, 1.570796, 1.930238],accel_mss,speed_ms,0,blend_radius_m)
    movel([0.360191, -1.287251, -2.631835, -0.793303, 1.570796, 1.930987],accel_mss,speed_ms,0,blend_radius_m)
    movel([0.360405, -1.287389, -2.631755, -0.793245, 1.570796, 1.931202],accel_mss,speed_ms,0,blend_radius_m)
    movel([0.360874, -1.287336, -2.631785, -0.793267, 1.570796, 1.931670],accel_mss,speed_ms,0,blend_radius_m)
    movel([0.361048, -1.287169, -2.631882, -0.793338, 1.570796, 1.931845],accel_mss,speed_ms,0,blend_radius_m)
    movel([0.361206, -1.286810, -2.632090, -0.793489, 1.570796, 1.932003],accel_mss,speed_ms,0,blend_radius_m)
    movel([0.361547, -1.285734, -2.632712, -0.793943, 1.570796, 1.932344],accel_mss,speed_ms,0,blend_radius_m)
    movel([0.362143, -1.283204, -2.634168, -0.795017, 1.570796, 1.932939],accel_mss,speed_ms,0,blend_radius_m)
    movel([0.362262, -1.281953, -2.634885, -0.795551, 1.570796, 1.933058],accel_mss,speed_ms,0,blend_radius_m)
    movel([0.362259, -1.279562, -2.636250, -0.796577, 1.570796, 1.933056],accel_mss,speed_ms,0,blend_radius_m)
    movel([0.362142, -1.278963, -2.636591, -0.796835, 1.570796, 1.932938],accel_mss,speed_ms,0,blend_radius_m)
    movel([0.361408, -1.277659, -2.637331, -0.797399, 1.570796, 1.932204],accel_mss,speed_ms,0,blend_radius_m)
    movel([0.360782, -1.276853, -2.637788, -0.797748, 1.570796, 1.931578],accel_mss,speed_ms,0,blend_radius_m)
    movel([0.360325, -1.276547, -2.637961, -0.797881, 1.570796, 1.931121],accel_mss,speed_ms,0,blend_radius_m)
    movel([0.359950, -1.276637, -2.637910, -0.797842, 1.570796, 1.930746],accel_mss,speed_ms,0,blend_radius_m)
    movel([0.359354, -1.277439, -2.637456, -0.797494, 1.570796, 1.930150],accel_mss,speed_ms,0,blend_radius_m)
    movel([0.357956, -1.276836, -2.637797, -0.797755, 1.570796, 1.928752],accel_mss,speed_ms,0,blend_radius_m)
    movel([0.357732, -1.276645, -2.637906, -0.797839, 1.570796, 1.928528],accel_mss,speed_ms,0,blend_radius_m)
    movel([0.357678, -1.276216, -2.638148, -0.798025, 1.570796, 1.928474],accel_mss,speed_ms,0,blend_radius_m)
    movel([0.357718, -1.276005, -2.638267, -0.798117, 1.570796, 1.928514],accel_mss,speed_ms,0,blend_radius_m)
    movel([0.357485, -1.275128, -2.638762, -0.798498, 1.570796, 1.928282],accel_mss,speed_ms,0,blend_radius_m)
    movel([0.357345, -1.274848, -2.638920, -0.798621, 1.570796, 1.928142],accel_mss,speed_ms,0,blend_radius_m)
    movel([0.357337, -1.274592, -2.639064, -0.798733, 1.570796, 1.928134],accel_mss,speed_ms,0,blend_radius_m)
    movel([0.358874, -1.274660, -2.639026, -0.798703, 1.570796, 1.929671],accel_mss,speed_ms,0,blend_radius_m)
    movel([0.359813, -1.274594, -2.639063, -0.798732, 1.570796, 1.930610],accel_mss,speed_ms,0,blend_radius_m)
    movel([0.360692, -1.274395, -2.639175, -0.798819, 1.570796, 1.931488],accel_mss,speed_ms,0,blend_radius_m)
    movel([0.361421, -1.274092, -2.639346, -0.798951, 1.570796, 1.932218],accel_mss,speed_ms,0,blend_radius_m)
    movel([0.361898, -1.273711, -2.639560, -0.799118, 1.570796, 1.932694],accel_mss,speed_ms,0,blend_radius_m)
    movel([0.362132, -1.273266, -2.639810, -0.799313, 1.570796, 1.932928],accel_mss,speed_ms,0,blend_radius_m)
    movel([0.362146, -1.272726, -2.640113, -0.799550, 1.570796, 1.932942],accel_mss,speed_ms,0,blend_radius_m)
    movel([0.361956, -1.272154, -2.640434, -0.799801, 1.570796, 1.932752],accel_mss,speed_ms,0,blend_radius_m)
    movel([0.361567, -1.271623, -2.640731, -0.800035, 1.570796, 1.932364],accel_mss,speed_ms,0,blend_radius_m)
    movel([0.361031, -1.271154, -2.640993, -0.800242, 1.570796, 1.931828],accel_mss,speed_ms,0,blend_radius_m)
    movel([0.359562, -1.270300, -2.641470, -0.800619, 1.570796, 1.930359],accel_mss,speed_ms,0,blend_radius_m)
    movel([0.359157, -1.270243, -2.641502, -0.800644, 1.570796, 1.929954],accel_mss,speed_ms,0,blend_radius_m)
    movel([0.359056, -1.270168, -2.641544, -0.800677, 1.570796, 1.929853],accel_mss,speed_ms,0,blend_radius_m)
    movel([0.360134, -1.268567, -2.642435, -0.801387, 1.570796, 1.930930],accel_mss,speed_ms,0,blend_radius_m)
    movel([0.360215, -1.268265, -2.642603, -0.801521, 1.570796, 1.931012],accel_mss,speed_ms,0,blend_radius_m)
    movel([0.360132, -1.267598, -2.642973, -0.801818, 1.570796, 1.930929],accel_mss,speed_ms,0,blend_radius_m)
    movel([0.360150, -1.267439, -2.643061, -0.801889, 1.570796, 1.930946],accel_mss,speed_ms,0,blend_radius_m)
    movel([0.360392, -1.267232, -2.643176, -0.801981, 1.570796, 1.931189],accel_mss,speed_ms,0,blend_radius_m)
    movel([0.360760, -1.266967, -2.643322, -0.802099, 1.570796, 1.931556],accel_mss,speed_ms,0,blend_radius_m)
    movel([0.361232, -1.266395, -2.643639, -0.802355, 1.570796, 1.932028],accel_mss,speed_ms,0,blend_radius_m)
    movel([0.361635, -1.265779, -2.643979, -0.802630, 1.570796, 1.932431],accel_mss,speed_ms,0,blend_radius_m)
    movel([0.361846, -1.265149, -2.644327, -0.802913, 1.570796, 1.932643],accel_mss,speed_ms,0,blend_radius_m)
    movel([0.361971, -1.264962, -2.644430, -0.802997, 1.570796, 1.932767],accel_mss,speed_ms,0,blend_radius_m)
    movel([0.362449, -1.264583, -2.644639, -0.803167, 1.570796, 1.933246],accel_mss,speed_ms,0,blend_radius_m)
    movel([0.363037, -1.264141, -2.644883, -0.803365, 1.570796, 1.933833],accel_mss,speed_ms,0,blend_radius_m)
    movel([0.363596, -1.263554, -2.645205, -0.803629, 1.570796, 1.934393],accel_mss,speed_ms,0,blend_radius_m)
    movel([0.364020, -1.262958, -2.645533, -0.803898, 1.570796, 1.934816],accel_mss,speed_ms,0,blend_radius_m)
    movel([0.364197, -1.262477, -2.645797, -0.804116, 1.570796, 1.934994],accel_mss,speed_ms,0,blend_radius_m)
    movel([0.364274, -1.262223, -2.645936, -0.804231, 1.570796, 1.935071],accel_mss,speed_ms,0,blend_radius_m)
    movel([0.364718, -1.261718, -2.646212, -0.804459, 1.570796, 1.935515],accel_mss,speed_ms,0,blend_radius_m)
    movel([0.365198, -1.261355, -2.646411, -0.804623, 1.570796, 1.935994],accel_mss,speed_ms,0,blend_radius_m)
    movel([0.366952, -1.260281, -2.646997, -0.805110, 1.570796, 1.937748],accel_mss,speed_ms,0,blend_radius_m)
    movel([0.368186, -1.259551, -2.647395, -0.805443, 1.570796, 1.938982],accel_mss,speed_ms,0,blend_radius_m)
    movel([0.369084, -1.258727, -2.647844, -0.805818, 1.570796, 1.939880],accel_mss,speed_ms,0,blend_radius_m)
    movel([0.369685, -1.257754, -2.648372, -0.806263, 1.570796, 1.940481],accel_mss,speed_ms,0,blend_radius_m)
    movel([0.370097, -1.256157, -2.649237, -0.806995, 1.570796, 1.940893],accel_mss,speed_ms,0,blend_radius_m)
    movel([0.370105, -1.255797, -2.649431, -0.807160, 1.570796, 1.940901],accel_mss,speed_ms,0,blend_radius_m)
    movel([0.369981, -1.255435, -2.649627, -0.807327, 1.570796, 1.940777],accel_mss,speed_ms,0,blend_radius_m)
    movel([0.369918, -1.255144, -2.649784, -0.807461, 1.570796, 1.940714],accel_mss,speed_ms,0,blend_radius_m)
    movel([0.370528, -1.255081, -2.649818, -0.807490, 1.570796, 1.941324],accel_mss,speed_ms,0,blend_radius_m)
    movel([0.371077, -1.255165, -2.649773, -0.807452, 1.570796, 1.941873],accel_mss,speed_ms,0,blend_radius_m)
    movel([0.372774, -1.254966, -2.649880, -0.807543, 1.570796, 1.943571],accel_mss,speed_ms,0,blend_radius_m)
    movel([0.373593, -1.254725, -2.650010, -0.807654, 1.570796, 1.944390],accel_mss,speed_ms,0,blend_radius_m)
    movel([0.374654, -1.254190, -2.650298, -0.807901, 1.570796, 1.945450],accel_mss,speed_ms,0,blend_radius_m)
    movel([0.375954, -1.253257, -2.650799, -0.808332, 1.570796, 1.946750],accel_mss,speed_ms,0,blend_radius_m)
    movel([0.377283, -1.252098, -2.651421, -0.808870, 1.570796, 1.948079],accel_mss,speed_ms,0,blend_radius_m)
    movel([0.378440, -1.250872, -2.652077, -0.809440, 1.570796, 1.949236],accel_mss,speed_ms,0,blend_radius_m)
    movel([0.379877, -1.249075, -2.653035, -0.810279, 1.570796, 1.950674],accel_mss,speed_ms,0,blend_radius_m)
    movel([0.382066, -1.246111, -2.654607, -0.811671, 1.570796, 1.952862],accel_mss,speed_ms,0,blend_radius_m)
    movel([0.386027, -1.240435, -2.657587, -0.814367, 1.570796, 1.956824],accel_mss,speed_ms,0,blend_radius_m)
    movel([0.388846, -1.235829, -2.659978, -0.816582, 1.570796, 1.959643],accel_mss,speed_ms,0,blend_radius_m)
    movel([0.389912, -1.233848, -2.660998, -0.817542, 1.570796, 1.960709],accel_mss,speed_ms,0,blend_radius_m)
    movel([0.390852, -1.231854, -2.662021, -0.818514, 1.570796, 1.961648],accel_mss,speed_ms,0,blend_radius_m)
    movel([0.392032, -1.228567, -2.663697, -0.820125, 1.570796, 1.962828],accel_mss,speed_ms,0,blend_radius_m)
    movel([0.392289, -1.227275, -2.664352, -0.820762, 1.570796, 1.963086],accel_mss,speed_ms,0,blend_radius_m)
    movel([0.392321, -1.226064, -2.664965, -0.821361, 1.570796, 1.963118],accel_mss,speed_ms,0,blend_radius_m)
    movel([0.392179, -1.225274, -2.665364, -0.821752, 1.570796, 1.962975],accel_mss,speed_ms,0,blend_radius_m)
    movel([0.391872, -1.224770, -2.665617, -0.822002, 1.570796, 1.962668],accel_mss,speed_ms,0,blend_radius_m)
    movel([0.391342, -1.224489, -2.665759, -0.822141, 1.570796, 1.962139],accel_mss,speed_ms,0,blend_radius_m)
    movel([0.389900, -1.224341, -2.665833, -0.822215, 1.570796, 1.960696],accel_mss,speed_ms,0,blend_radius_m)
    movel([0.389715, -1.224255, -2.665876, -0.822257, 1.570796, 1.960512],accel_mss,speed_ms,0,blend_radius_m)
    movel([0.389854, -1.223612, -2.666200, -0.822578, 1.570796, 1.960651],accel_mss,speed_ms,0,blend_radius_m)
    movel([0.390072, -1.223166, -2.666424, -0.822800, 1.570796, 1.960868],accel_mss,speed_ms,0,blend_radius_m)
    movel([0.394222, -1.216131, -2.669925, -0.826333, 1.570796, 1.965019],accel_mss,speed_ms,0,blend_radius_m)
    movel([0.395044, -1.214444, -2.670756, -0.827189, 1.570796, 1.965841],accel_mss,speed_ms,0,blend_radius_m)
    movel([0.396231, -1.211292, -2.672300, -0.828796, 1.570796, 1.967027],accel_mss,speed_ms,0,blend_radius_m)
    movel([0.396582, -1.209851, -2.673003, -0.829535, 1.570796, 1.967378],accel_mss,speed_ms,0,blend_radius_m)
    movel([0.396736, -1.208646, -2.673589, -0.830154, 1.570796, 1.967532],accel_mss,speed_ms,0,blend_radius_m)
    movel([0.396696, -1.207523, -2.674133, -0.830733, 1.570796, 1.967492],accel_mss,speed_ms,0,blend_radius_m)
    movel([0.396442, -1.206554, -2.674602, -0.831234, 1.570796, 1.967238],accel_mss,speed_ms,0,blend_radius_m)
    movel([0.395927, -1.205666, -2.675030, -0.831693, 1.570796, 1.966723],accel_mss,speed_ms,0,blend_radius_m)
    movel([0.395237, -1.204971, -2.675365, -0.832054, 1.570796, 1.966033],accel_mss,speed_ms,0,blend_radius_m)
    movel([0.394452, -1.204583, -2.675551, -0.832255, 1.570796, 1.965249],accel_mss,speed_ms,0,blend_radius_m)
    movel([0.393065, -1.204447, -2.675617, -0.832326, 1.570796, 1.963861],accel_mss,speed_ms,0,blend_radius_m)
    movel([0.391506, -1.204756, -2.675468, -0.832165, 1.570796, 1.962302],accel_mss,speed_ms,0,blend_radius_m)
    movel([0.390152, -1.205407, -2.675155, -0.831827, 1.570796, 1.960948],accel_mss,speed_ms,0,blend_radius_m)
    movel([0.389698, -1.205785, -2.674972, -0.831632, 1.570796, 1.960495],accel_mss,speed_ms,0,blend_radius_m)
    movel([0.389359, -1.206257, -2.674745, -0.831387, 1.570796, 1.960156],accel_mss,speed_ms,0,blend_radius_m)
    movel([0.389256, -1.206631, -2.674564, -0.831194, 1.570796, 1.960052],accel_mss,speed_ms,0,blend_radius_m)
    movel([0.389401, -1.206791, -2.674487, -0.831111, 1.570796, 1.960198],accel_mss,speed_ms,0,blend_radius_m)
    movel([0.389823, -1.206713, -2.674525, -0.831152, 1.570796, 1.960619],accel_mss,speed_ms,0,blend_radius_m)
    movel([0.390548, -1.206367, -2.674692, -0.831331, 1.570796, 1.961344],accel_mss,speed_ms,0,blend_radius_m)
    movel([0.391369, -1.206002, -2.674868, -0.831519, 1.570796, 1.962165],accel_mss,speed_ms,0,blend_radius_m)
    movel([0.392170, -1.205793, -2.674969, -0.831628, 1.570796, 1.962966],accel_mss,speed_ms,0,blend_radius_m)
    movel([0.392910, -1.205753, -2.674988, -0.831648, 1.570796, 1.963706],accel_mss,speed_ms,0,blend_radius_m)
    movel([0.393555, -1.205887, -2.674923, -0.831579, 1.570796, 1.964352],accel_mss,speed_ms,0,blend_radius_m)
    movel([0.394102, -1.206189, -2.674777, -0.831422, 1.570796, 1.964898],accel_mss,speed_ms,0,blend_radius_m)
    movel([0.394505, -1.206646, -2.674557, -0.831186, 1.570796, 1.965302],accel_mss,speed_ms,0,blend_radius_m)
    movel([0.394770, -1.207247, -2.674266, -0.830876, 1.570796, 1.965566],accel_mss,speed_ms,0,blend_radius_m)
    movel([0.394864, -1.208674, -2.673575, -0.830140, 1.570796, 1.965661],accel_mss,speed_ms,0,blend_radius_m)
    movel([0.394753, -1.209359, -2.673242, -0.829788, 1.570796, 1.965550],accel_mss,speed_ms,0,blend_radius_m)
    movel([0.393999, -1.211673, -2.672115, -0.828602, 1.570796, 1.964796],accel_mss,speed_ms,0,blend_radius_m)
    movel([0.393069, -1.213993, -2.670977, -0.827418, 1.570796, 1.963866],accel_mss,speed_ms,0,blend_radius_m)
    movel([0.392028, -1.216117, -2.669932, -0.826340, 1.570796, 1.962824],accel_mss,speed_ms,0,blend_radius_m)
    movel([0.390762, -1.218270, -2.668866, -0.825253, 1.570796, 1.961559],accel_mss,speed_ms,0,blend_radius_m)
    movel([0.389150, -1.220668, -2.667673, -0.824048, 1.570796, 1.959947],accel_mss,speed_ms,0,blend_radius_m)
    movel([0.387454, -1.223238, -2.666388, -0.822764, 1.570796, 1.958250],accel_mss,speed_ms,0,blend_radius_m)
    movel([0.387029, -1.224046, -2.665981, -0.822361, 1.570796, 1.957825],accel_mss,speed_ms,0,blend_radius_m)
    movel([0.386745, -1.224845, -2.665579, -0.821964, 1.570796, 1.957541],accel_mss,speed_ms,0,blend_radius_m)
    movel([0.386633, -1.225555, -2.665221, -0.821612, 1.570796, 1.957429],accel_mss,speed_ms,0,blend_radius_m)
    movel([0.386687, -1.226197, -2.664898, -0.821295, 1.570796, 1.957483],accel_mss,speed_ms,0,blend_radius_m)
    movel([0.387662, -1.228824, -2.663567, -0.819999, 1.570796, 1.958458],accel_mss,speed_ms,0,blend_radius_m)
    movel([0.387854, -1.229743, -2.663099, -0.819547, 1.570796, 1.958651],accel_mss,speed_ms,0,blend_radius_m)
    movel([0.387852, -1.230708, -2.662607, -0.819074, 1.570796, 1.958648],accel_mss,speed_ms,0,blend_radius_m)
    movel([0.387665, -1.231869, -2.662014, -0.818507, 1.570796, 1.958462],accel_mss,speed_ms,0,blend_radius_m)
    movel([0.387304, -1.233122, -2.661371, -0.817896, 1.570796, 1.958100],accel_mss,speed_ms,0,blend_radius_m)
    movel([0.386773, -1.234398, -2.660716, -0.817275, 1.570796, 1.957570],accel_mss,speed_ms,0,blend_radius_m)
    movel([0.385075, -1.237477, -2.659125, -0.815786, 1.570796, 1.955871],accel_mss,speed_ms,0,blend_radius_m)
    movel([0.382546, -1.241184, -2.657196, -0.814009, 1.570796, 1.953343],accel_mss,speed_ms,0,blend_radius_m)
    movel([0.379075, -1.245664, -2.654842, -0.811882, 1.570796, 1.949871],accel_mss,speed_ms,0,blend_radius_m)
    movel([0.377241, -1.247936, -2.653640, -0.810813, 1.570796, 1.948038],accel_mss,speed_ms,0,blend_radius_m)
    movel([0.377299, -1.246963, -2.654156, -0.811270, 1.570796, 1.948095],accel_mss,speed_ms,0,blend_radius_m)
    movel([0.377210, -1.246132, -2.654596, -0.811662, 1.570796, 1.948006],accel_mss,speed_ms,0,blend_radius_m)
    movel([0.376813, -1.245750, -2.654797, -0.811842, 1.570796, 1.947609],accel_mss,speed_ms,0,blend_radius_m)
    movel([0.375902, -1.245677, -2.654836, -0.811876, 1.570796, 1.946698],accel_mss,speed_ms,0,blend_radius_m)
    movel([0.370601, -1.246296, -2.654509, -0.811585, 1.570796, 1.941397],accel_mss,speed_ms,0,blend_radius_m)
    movel([0.371302, -1.245620, -2.654866, -0.811903, 1.570796, 1.942098],accel_mss,speed_ms,0,blend_radius_m)
    movel([0.371929, -1.244876, -2.655258, -0.812255, 1.570796, 1.942726],accel_mss,speed_ms,0,blend_radius_m)
    movel([0.372160, -1.244462, -2.655476, -0.812451, 1.570796, 1.942957],accel_mss,speed_ms,0,blend_radius_m)
    movel([0.372565, -1.243372, -2.656049, -0.812967, 1.570796, 1.943362],accel_mss,speed_ms,0,blend_radius_m)
    movel([0.372598, -1.243000, -2.656245, -0.813144, 1.570796, 1.943394],accel_mss,speed_ms,0,blend_radius_m)
    movel([0.372147, -1.242129, -2.656702, -0.813559, 1.570796, 1.942943],accel_mss,speed_ms,0,blend_radius_m)
    movel([0.371192, -1.241262, -2.657155, -0.813972, 1.570796, 1.941988],accel_mss,speed_ms,0,blend_radius_m)
    movel([0.369777, -1.240716, -2.657441, -0.814233, 1.570796, 1.940574],accel_mss,speed_ms,0,blend_radius_m)
    movel([0.368124, -1.240545, -2.657530, -0.814314, 1.570796, 1.938921],accel_mss,speed_ms,0,blend_radius_m)
    movel([0.366461, -1.240805, -2.657394, -0.814190, 1.570796, 1.937258],accel_mss,speed_ms,0,blend_radius_m)
    movel([0.365983, -1.240950, -2.657318, -0.814121, 1.570796, 1.936779],accel_mss,speed_ms,0,blend_radius_m)
    movel([0.364436, -1.241601, -2.656978, -0.813810, 1.570796, 1.935232],accel_mss,speed_ms,0,blend_radius_m)
    movel([0.364269, -1.241642, -2.656956, -0.813790, 1.570796, 1.935066],accel_mss,speed_ms,0,blend_radius_m)
    movel([0.364262, -1.241368, -2.657100, -0.813921, 1.570796, 1.935059],accel_mss,speed_ms,0,blend_radius_m)
    movel([0.364210, -1.241166, -2.657205, -0.814017, 1.570796, 1.935006],accel_mss,speed_ms,0,blend_radius_m)
    movel([0.363872, -1.241127, -2.657226, -0.814036, 1.570796, 1.934668],accel_mss,speed_ms,0,blend_radius_m)
    movel([0.363306, -1.241256, -2.657158, -0.813975, 1.570796, 1.934103],accel_mss,speed_ms,0,blend_radius_m)
    movel([0.362134, -1.241737, -2.656907, -0.813745, 1.570796, 1.932930],accel_mss,speed_ms,0,blend_radius_m)
    movel([0.361852, -1.241781, -2.656884, -0.813724, 1.570796, 1.932648],accel_mss,speed_ms,0,blend_radius_m)
    movel([0.361186, -1.241414, -2.657076, -0.813899, 1.570796, 1.931983],accel_mss,speed_ms,0,blend_radius_m)
    movel([0.360348, -1.240959, -2.657314, -0.814117, 1.570796, 1.931144],accel_mss,speed_ms,0,blend_radius_m)
    movel([0.359290, -1.240700, -2.657449, -0.814240, 1.570796, 1.930086],accel_mss,speed_ms,0,blend_radius_m)
    movel([0.358043, -1.240645, -2.657477, -0.814266, 1.570796, 1.928839],accel_mss,speed_ms,0,blend_radius_m)
    movel([0.356641, -1.240796, -2.657398, -0.814194, 1.570796, 1.927437],accel_mss,speed_ms,0,blend_radius_m)
    movel([0.356107, -1.240985, -2.657300, -0.814104, 1.570796, 1.926904],accel_mss,speed_ms,0,blend_radius_m)
    movel([0.355823, -1.241301, -2.657135, -0.813953, 1.570796, 1.926619],accel_mss,speed_ms,0,blend_radius_m)
    movel([0.355802, -1.241738, -2.656906, -0.813745, 1.570796, 1.926598],accel_mss,speed_ms,0,blend_radius_m)
    movel([0.356089, -1.242314, -2.656605, -0.813471, 1.570796, 1.926885],accel_mss,speed_ms,0,blend_radius_m)
    movel([0.356286, -1.242634, -2.656437, -0.813318, 1.570796, 1.927082],accel_mss,speed_ms,0,blend_radius_m)
    movel([0.356767, -1.243795, -2.655827, -0.812767, 1.570796, 1.927563],accel_mss,speed_ms,0,blend_radius_m)
    movel([0.356718, -1.244002, -2.655719, -0.812669, 1.570796, 1.927514],accel_mss,speed_ms,0,blend_radius_m)
    movel([0.356084, -1.244710, -2.655346, -0.812333, 1.570796, 1.926880],accel_mss,speed_ms,0,blend_radius_m)
    movel([0.355318, -1.245463, -2.654948, -0.811977, 1.570796, 1.926114],accel_mss,speed_ms,0,blend_radius_m)
    movel([0.355372, -1.242031, -2.656753, -0.813605, 1.570796, 1.926168],accel_mss,speed_ms,0,blend_radius_m)
    movel([0.355267, -1.241514, -2.657023, -0.813851, 1.570796, 1.926064],accel_mss,speed_ms,0,blend_radius_m)
    movel([0.354972, -1.241369, -2.657099, -0.813921, 1.570796, 1.925768],accel_mss,speed_ms,0,blend_radius_m)
    movel([0.354922, -1.241215, -2.657180, -0.813994, 1.570796, 1.925718],accel_mss,speed_ms,0,blend_radius_m)
    movel([0.355008, -1.240323, -2.657646, -0.814420, 1.570796, 1.925804],accel_mss,speed_ms,0,blend_radius_m)
    movel([0.355006, -1.239953, -2.657838, -0.814598, 1.570796, 1.925803],accel_mss,speed_ms,0,blend_radius_m)
    movel([0.354631, -1.238534, -2.658577, -0.815278, 1.570796, 1.925427],accel_mss,speed_ms,0,blend_radius_m)
    movel([0.354664, -1.238252, -2.658723, -0.815414, 1.570796, 1.925460],accel_mss,speed_ms,0,blend_radius_m)
    movel([0.354797, -1.238134, -2.658785, -0.815471, 1.570796, 1.925593],accel_mss,speed_ms,0,blend_radius_m)
    movel([0.358831, -1.239922, -2.657855, -0.814612, 1.570796, 1.929627],accel_mss,speed_ms,0,blend_radius_m)
    movel([0.359202, -1.239939, -2.657846, -0.814604, 1.570796, 1.929998],accel_mss,speed_ms,0,blend_radius_m)
    movel([0.359517, -1.239789, -2.657924, -0.814676, 1.570796, 1.930314],accel_mss,speed_ms,0,blend_radius_m)
    movel([0.359744, -1.239554, -2.658046, -0.814789, 1.570796, 1.930541],accel_mss,speed_ms,0,blend_radius_m)
    movel([0.359869, -1.239025, -2.658321, -0.815042, 1.570796, 1.930665],accel_mss,speed_ms,0,blend_radius_m)
    movel([0.359789, -1.238428, -2.658632, -0.815329, 1.570796, 1.930586],accel_mss,speed_ms,0,blend_radius_m)
    movel([0.359186, -1.236532, -2.659615, -0.816242, 1.570796, 1.929982],accel_mss,speed_ms,0,blend_radius_m)
    movel([0.358683, -1.235665, -2.660063, -0.816661, 1.570796, 1.929479],accel_mss,speed_ms,0,blend_radius_m)
    movel([0.357804, -1.234609, -2.660607, -0.817173, 1.570796, 1.928601],accel_mss,speed_ms,0,blend_radius_m)
    movel([0.357601, -1.234272, -2.660781, -0.817337, 1.570796, 1.928397],accel_mss,speed_ms,0,blend_radius_m)
    movel([0.357424, -1.233056, -2.661405, -0.817927, 1.570796, 1.928221],accel_mss,speed_ms,0,blend_radius_m)
    movel([0.357082, -1.232635, -2.661621, -0.818133, 1.570796, 1.927879],accel_mss,speed_ms,0,blend_radius_m)
    movel([0.356444, -1.232400, -2.661741, -0.818247, 1.570796, 1.927240],accel_mss,speed_ms,0,blend_radius_m)
    movel([0.355670, -1.232385, -2.661749, -0.818255, 1.570796, 1.926467],accel_mss,speed_ms,0,blend_radius_m)
    movel([0.354500, -1.232614, -2.661632, -0.818143, 1.570796, 1.925296],accel_mss,speed_ms,0,blend_radius_m)
    movel([0.353288, -1.233034, -2.661416, -0.817938, 1.570796, 1.924084],accel_mss,speed_ms,0,blend_radius_m)
    movel([0.350182, -1.234547, -2.660639, -0.817203, 1.570796, 1.920979],accel_mss,speed_ms,0,blend_radius_m)
    movel([0.348019, -1.235864, -2.659960, -0.816565, 1.570796, 1.918815],accel_mss,speed_ms,0,blend_radius_m)
    movel([0.342224, -1.239942, -2.657844, -0.814603, 1.570796, 1.913020],accel_mss,speed_ms,0,blend_radius_m)
    movel([0.340538, -1.241338, -2.657116, -0.813936, 1.570796, 1.911335],accel_mss,speed_ms,0,blend_radius_m)
    movel([0.339435, -1.242459, -2.656529, -0.813402, 1.570796, 1.910231],accel_mss,speed_ms,0,blend_radius_m)
    movel([0.338884, -1.243080, -2.656203, -0.813106, 1.570796, 1.909680],accel_mss,speed_ms,0,blend_radius_m)
    movel([0.337893, -1.244436, -2.655490, -0.812463, 1.570796, 1.908689],accel_mss,speed_ms,0,blend_radius_m)
    movel([0.337454, -1.245258, -2.655057, -0.812074, 1.570796, 1.908251],accel_mss,speed_ms,0,blend_radius_m)
    movel([0.335224, -1.250919, -2.652052, -0.809418, 1.570796, 1.906020],accel_mss,speed_ms,0,blend_radius_m)
    movel([0.334551, -1.252554, -2.651177, -0.808659, 1.570796, 1.905348],accel_mss,speed_ms,0,blend_radius_m)
    movel([0.333515, -1.254791, -2.649974, -0.807624, 1.570796, 1.904311],accel_mss,speed_ms,0,blend_radius_m)
    movel([0.332477, -1.256480, -2.649062, -0.806847, 1.570796, 1.903273],accel_mss,speed_ms,0,blend_radius_m)
    movel([0.331180, -1.258227, -2.648116, -0.806047, 1.570796, 1.901976],accel_mss,speed_ms,0,blend_radius_m)
    movel([0.329636, -1.260022, -2.647138, -0.805228, 1.570796, 1.900433],accel_mss,speed_ms,0,blend_radius_m)
    movel([0.327848, -1.261859, -2.646135, -0.804395, 1.570796, 1.898644],accel_mss,speed_ms,0,blend_radius_m)
    movel([0.325480, -1.264317, -2.644786, -0.803286, 1.570796, 1.896276],accel_mss,speed_ms,0,blend_radius_m)
    movel([0.324722, -1.265235, -2.644280, -0.802874, 1.570796, 1.895518],accel_mss,speed_ms,0,blend_radius_m)
    movel([0.324068, -1.266194, -2.643750, -0.802445, 1.570796, 1.894864],accel_mss,speed_ms,0,blend_radius_m)
    movel([0.322959, -1.268375, -2.642541, -0.801472, 1.570796, 1.893755],accel_mss,speed_ms,0,blend_radius_m)
    movel([0.321541, -1.272110, -2.640458, -0.799821, 1.570796, 1.892337],accel_mss,speed_ms,0,blend_radius_m)
    movel([0.320732, -1.274531, -2.639099, -0.798759, 1.570796, 1.891528],accel_mss,speed_ms,0,blend_radius_m)
    movel([0.320752, -1.274802, -2.638946, -0.798641, 1.570796, 1.891548],accel_mss,speed_ms,0,blend_radius_m)
    movel([0.321115, -1.274882, -2.638901, -0.798606, 1.570796, 1.891911],accel_mss,speed_ms,0,blend_radius_m)
    movel([0.321292, -1.274809, -2.638942, -0.798638, 1.570796, 1.892088],accel_mss,speed_ms,0,blend_radius_m)
    movel([0.321590, -1.274542, -2.639093, -0.798755, 1.570796, 1.892387],accel_mss,speed_ms,0,blend_radius_m)
    movel([0.321738, -1.274280, -2.639240, -0.798869, 1.570796, 1.892534],accel_mss,speed_ms,0,blend_radius_m)
    movel([0.323140, -1.270782, -2.641201, -0.800406, 1.570796, 1.893936],accel_mss,speed_ms,0,blend_radius_m)
    movel([0.323671, -1.269422, -2.641960, -0.801008, 1.570796, 1.894467],accel_mss,speed_ms,0,blend_radius_m)
    movel([0.324926, -1.266563, -2.643546, -0.802280, 1.570796, 1.895723],accel_mss,speed_ms,0,blend_radius_m)
    movel([0.325554, -1.265645, -2.644054, -0.802691, 1.570796, 1.896351],accel_mss,speed_ms,0,blend_radius_m)
    movel([0.327476, -1.263458, -2.645258, -0.803673, 1.570796, 1.898272],accel_mss,speed_ms,0,blend_radius_m)
    movel([0.328937, -1.262004, -2.646055, -0.804329, 1.570796, 1.899733],accel_mss,speed_ms,0,blend_radius_m)
    movel([0.331625, -1.259206, -2.647583, -0.805600, 1.570796, 1.902421],accel_mss,speed_ms,0,blend_radius_m)
    movel([0.332584, -1.257969, -2.648255, -0.806164, 1.570796, 1.903380],accel_mss,speed_ms,0,blend_radius_m)
    movel([0.334432, -1.255148, -2.649782, -0.807459, 1.570796, 1.905229],accel_mss,speed_ms,0,blend_radius_m)
    movel([0.334955, -1.254144, -2.650322, -0.807922, 1.570796, 1.905751],accel_mss,speed_ms,0,blend_radius_m)
    movel([0.337916, -1.246661, -2.654316, -0.811412, 1.570796, 1.908713],accel_mss,speed_ms,0,blend_radius_m)
    movel([0.338858, -1.244774, -2.655312, -0.812303, 1.570796, 1.909654],accel_mss,speed_ms,0,blend_radius_m)
    movel([0.339889, -1.243369, -2.656051, -0.812969, 1.570796, 1.910685],accel_mss,speed_ms,0,blend_radius_m)
    movel([0.341379, -1.241886, -2.656829, -0.813674, 1.570796, 1.912175],accel_mss,speed_ms,0,blend_radius_m)
